
// ===== library: MasterCopy "GB2312_TO_UTF8" =====

// folder: FB/GB2312_UTF8

FUNCTION_BLOCK "GB2312_TO_UTF8"   // FB8, SCL
{ S7_Optimized_Access := 'TRUE' }
VERSION : 0.1
   VAR_INPUT
      GB2312 : String[254];
   END_VAR
   VAR_OUTPUT
      UTF8 : String[254];
   END_VAR
   VAR
      g_u : "GB2_TO_UNI";
      u_u8 : "UNI_TO_UTF8";
   END_VAR
   VAR_TEMP
      i : UDInt;
      j : UDInt;
      lenGB2 : Int;
      tempword : Word;
      tempstr : String[4];
   END_VAR
BEGIN
   #UTF8 := '';
   #lenGB2 := LEN(#GB2312);
   IF #lenGB2 > 0 THEN
       #j := 1;
       FOR #i := 1 TO INT_TO_UDINT(#lenGB2) DO
           IF #i = #j THEN
               IF BYTE_TO_WORD(#GB2312[#i]) < 16#0080 THEN
                   #tempword := BYTE_TO_WORD(#GB2312[#i]);
                   #j := #j + 1;
               ELSE
                   #tempword := BYTE_TO_WORD(#GB2312[#i]);
                   #tempword := SHL(IN := #tempword, N := 8);
                   #tempword := #tempword OR BYTE_TO_WORD(#GB2312[#i + 1]);
                   #j := #j + 2;
               END_IF;
               #g_u(GB2312 := #tempword,
                    UNICODE => #tempword);
               #u_u8(UNICODE := #tempword,
                     UTF8 => #tempstr);
               #UTF8 := CONCAT(IN1 := #UTF8, IN2 := #tempstr);
           END_IF;
       END_FOR;
   END_IF;
END_FUNCTION_BLOCK

// ===== library: MasterCopy "UTF8_TO_GB2312" =====

// folder: FB/GB2312_UTF8

FUNCTION_BLOCK "UTF8_TO_GB2312"   // FB10, SCL
{ S7_Optimized_Access := 'TRUE' }
VERSION : 0.1
   VAR_INPUT
      UTF8 : String[254];
   END_VAR
   VAR_OUTPUT
      GB2312 : String[254];
   END_VAR
   VAR
      u8_u : "UTF8_TO_UNI";
      u_g : "UNI_TO_GB2";
   END_VAR
   VAR_TEMP
      i : Int;
      j : Int;
      lenUTF8 : Int;
      tempword : Word;
      tempstr : String[5];
   END_VAR
BEGIN
   #GB2312 := '';
   #tempstr := '0000';
   #lenUTF8 := LEN(#UTF8);
   IF #lenUTF8 > 0 THEN
       #j := 1;
       FOR #i := 1 TO #lenUTF8 DO
           IF #i = #j THEN
               IF BYTE_TO_WORD(#UTF8[#i]) < 16#0080 THEN
                   #tempstr := MID(IN := #UTF8, L := 1, P := #i);
                   #j := #j + 1;
               ELSIF BYTE_TO_WORD(#UTF8[#i]) >= 16#C0 AND BYTE_TO_WORD(#UTF8[#i]) < 16#E0 THEN
                   #tempstr := MID(IN := #UTF8, L := 2, P := #i);
                   #j := #j + 2;
               ELSIF BYTE_TO_WORD(#UTF8[#i]) >= 16#E0 AND BYTE_TO_WORD(#UTF8[#i]) < 16#F0 THEN
                   #tempstr := MID(IN := #UTF8, L := 3, P := #i);
                   #j := #j + 3;
               ELSIF BYTE_TO_WORD(#UTF8[#i]) >= 16#F0 AND BYTE_TO_WORD(#UTF8[#i]) < 16#F8 THEN
                   #tempstr := MID(IN := #UTF8, L := 4, P := #i);
                   #j := #j + 4;
               END_IF;
               IF BYTE_TO_WORD(#UTF8[#i]) >= 16#0080 THEN
                   #u8_u(UTF8 := #tempstr,
                         UNICODE => #tempword);
                   #u_g(UNICODE := #tempword,
                        GB2312 => #tempword);
                   #tempstr[2] := WORD_TO_BYTE(#tempword AND 16#FF);
                   #tempstr[1] := WORD_TO_BYTE(SHR(IN := #tempword, N := 8) AND 16#FF);
                   #tempstr := LEFT(IN := #tempstr, L := 2);
               END_IF;
               #GB2312 := CONCAT(IN1 := #GB2312, IN2 := #tempstr);
           END_IF;
       END_FOR;
   END_IF;
END_FUNCTION_BLOCK

// ===== library: MasterCopy "GB2312_TO_UTF16" =====

// folder: FB/GB2312_UTF16

FUNCTION_BLOCK "GB2312_TO_UTF16"   // FB13, SCL
{ S7_Optimized_Access := 'TRUE' }
VERSION : 0.1
   VAR_INPUT
      GB2312 : String[254];
   END_VAR
   VAR_OUTPUT
      UTF16 : WString;
   END_VAR
   VAR
      g_u : "GB2_TO_UNI";
   END_VAR
   VAR_TEMP
      i : UDInt;
      j : UDInt;
      lenGB2 : Int;
      tempword : Word;
      tempWstr : WString[4];
   END_VAR
BEGIN
   #UTF16 := WSTRING#'';
   #tempWstr := WSTRING#'0000';
   #lenGB2 := LEN(#GB2312);
   IF #lenGB2 > 0 THEN
       #j := 1;
       FOR #i := 1 TO INT_TO_UDINT(#lenGB2) DO
           IF #i = #j THEN
               IF BYTE_TO_WORD(#GB2312[#i]) < 16#0080 THEN
                   #tempword := BYTE_TO_WORD(#GB2312[#i]);
                   #j := #j + 1;
               ELSE
                   #tempword := BYTE_TO_WORD(#GB2312[#i]);
                   #tempword := SHL(IN := #tempword, N := 8);
                   #tempword := #tempword OR BYTE_TO_WORD(#GB2312[#i + 1]);
                   #j := #j + 2;
               END_IF;
               #g_u(GB2312 := #tempword,
                    UNICODE => #tempword);
               #tempWstr[1] := #tempword;
               #tempWstr := LEFT(IN := #tempWstr, L := 1);
               #UTF16 := CONCAT(IN1 := #UTF16, IN2 := #tempWstr);
           END_IF;
       END_FOR;
   END_IF;
END_FUNCTION_BLOCK

// ===== library: MasterCopy "UTF16_TO_GB2312" =====

// folder: FB/GB2312_UTF16

FUNCTION_BLOCK "UTF16_TO_GB2312"   // FB11, SCL
{ S7_Optimized_Access := 'TRUE' }
VERSION : 0.1
   VAR_INPUT
      UTF16 : WString;
   END_VAR
   VAR_OUTPUT
      GB2312 : String[254];
   END_VAR
   VAR
      u_g : "UNI_TO_GB2";
   END_VAR
   VAR_TEMP
      i : Int;
      j : Int;
      lenUTF16 : Int;
      tempword : Word;
      tempstr : String[5];
   END_VAR
BEGIN
   #GB2312 := '';
   #tempstr := '0000';
   #lenUTF16 := LEN(#UTF16);
   IF #lenUTF16 > 0 THEN
       #j := 1;
       FOR #i := 1 TO #lenUTF16 DO
           #tempword := WCHAR_TO_WORD(#UTF16[#i]);
           IF #tempword < 16#0080 THEN
               #tempstr[1] := WORD_TO_BYTE(#tempword);
               #tempstr := LEFT(IN := #tempstr, L := 1);
           END_IF;
           IF #tempword >= 16#0080 THEN
               #u_g(UNICODE := #tempword,
                    GB2312 => #tempword);
               #tempstr[2] := WORD_TO_BYTE(#tempword AND 16#FF);
               #tempstr[1] := WORD_TO_BYTE(SHR(IN := #tempword, N := 8) AND 16#FF);
               #tempstr := LEFT(IN := #tempstr, L := 2);
           END_IF;
           #GB2312 := CONCAT(IN1 := #GB2312, IN2 := #tempstr);
       END_FOR;
   END_IF;
END_FUNCTION_BLOCK

// ===== library: MasterCopy "WStr_TO_Str_x4" =====

// folder: FB/GB2312_UTF16

FUNCTION_BLOCK "WStr_TO_Str_x4"   // FB12, SCL
{ S7_Optimized_Access := 'TRUE' }
VERSION : 0.1
   VAR_INPUT
      X0_Wstr : WString;
      X1_Wstr : WString;
      X2_Wstr : WString;
      X3_Wstr : WString;
   END_VAR
   VAR_OUTPUT
      X0_Str : String;
      X1_Str : String;
      X2_Str : String;
      X3_Str : String;
   END_VAR
   VAR
      U16_gb2 : "UTF16_TO_GB2312";
   END_VAR
   VAR_TEMP
      i : Int;
      j : Int;
      lenUTF16 : Int;
      tempword : Word;
      tempstr : String[5];
   END_VAR
BEGIN
   #U16_gb2(UTF16 := #X0_Wstr,
            GB2312 => #X0_Str);
   #U16_gb2(UTF16 := #X1_Wstr,
            GB2312 => #X1_Str);
   #U16_gb2(UTF16 := #X2_Wstr,
            GB2312 => #X2_Str);
   #U16_gb2(UTF16 := #X3_Wstr,
            GB2312 => #X3_Str);
END_FUNCTION_BLOCK

// ===== library: MasterCopy "UTF8_TO_GBK" =====

// folder: FB/GBK_UTF8

FUNCTION_BLOCK "UTF8_TO_GBK"   // FB6, SCL
{ S7_Optimized_Access := 'TRUE' }
VERSION : 0.1
   VAR_INPUT
      UTF8 : String[254];
   END_VAR
   VAR_OUTPUT
      GBK : String[254];
   END_VAR
   VAR
      u8_u : "UTF8_TO_UNI";
      u_g : "UNI_TO_GBK";
   END_VAR
   VAR_TEMP
      i : Int;
      j : Int;
      lenUTF8 : Int;
      tempword : Word;
      tempstr : String[5];
   END_VAR
BEGIN
   #GBK := '';
   #tempstr := '0000';
   #lenUTF8 := LEN(#UTF8);
   IF #lenUTF8 > 0 THEN
       #j := 1;
       FOR #i := 1 TO #lenUTF8 DO
           IF #i = #j THEN
               IF BYTE_TO_WORD(#UTF8[#i]) < 16#0080 THEN
                   #tempstr := MID(IN := #UTF8, L := 1, P := #i);
                   #j := #j + 1;
               ELSIF BYTE_TO_WORD(#UTF8[#i]) >= 16#C0 AND BYTE_TO_WORD(#UTF8[#i]) < 16#E0 THEN
                   #tempstr := MID(IN := #UTF8, L := 2, P := #i);
                   #j := #j + 2;
               ELSIF BYTE_TO_WORD(#UTF8[#i]) >= 16#E0 AND BYTE_TO_WORD(#UTF8[#i]) < 16#F0 THEN
                   #tempstr := MID(IN := #UTF8, L := 3, P := #i);
                   #j := #j + 3;
               ELSIF BYTE_TO_WORD(#UTF8[#i]) >= 16#F0 AND BYTE_TO_WORD(#UTF8[#i]) < 16#F8 THEN
                   #tempstr := MID(IN := #UTF8, L := 4, P := #i);
                   #j := #j + 4;
               END_IF;
               IF BYTE_TO_WORD(#UTF8[#i]) >= 16#0080 THEN
                   #u8_u(UTF8 := #tempstr,
                         UNICODE => #tempword);
                   #u_g(UNICODE := #tempword,
                        GBK => #tempword);
                   #tempstr[2] := WORD_TO_BYTE(#tempword AND 16#FF);
                   #tempstr[1] := WORD_TO_BYTE(SHR(IN := #tempword, N := 8) AND 16#FF);
                   #tempstr := LEFT(IN := #tempstr, L := 2);
               END_IF;
               #GBK := CONCAT(IN1 := #GBK, IN2 := #tempstr);
           END_IF;
       END_FOR;
   END_IF;
END_FUNCTION_BLOCK

// ===== library: MasterCopy "GBK_TO_UTF8" =====

// folder: FB/GBK_UTF8

FUNCTION_BLOCK "GBK_TO_UTF8"   // FB5, SCL
{ S7_Optimized_Access := 'TRUE' }
VERSION : 0.1
   VAR_INPUT
      GBK : String[254];
   END_VAR
   VAR_OUTPUT
      UTF8 : String[254];
   END_VAR
   VAR
      g_u : "GBK_TO_UNI";
      u_u8 : "UNI_TO_UTF8";
   END_VAR
   VAR_TEMP
      i : UDInt;
      j : UDInt;
      lenGBK : Int;
      tempword : Word;
      tempstr : String[4];
   END_VAR
BEGIN
   #UTF8 := '';
   #lenGBK := LEN(#GBK);
   IF #lenGBK > 0 THEN
       #j := 1;
       FOR #i := 1 TO INT_TO_UDINT(#lenGBK) DO
           IF #i = #j THEN
               IF BYTE_TO_WORD(#GBK[#i]) < 16#0080 THEN
                   #tempword := BYTE_TO_WORD(#GBK[#i]);
                   #j := #j + 1;
               ELSE
                   #tempword := BYTE_TO_WORD(#GBK[#i]);
                   #tempword := SHL(IN := #tempword, N:=8);
                   #tempword := #tempword OR BYTE_TO_WORD(#GBK[#i + 1]);
                   #j := #j + 2;
               END_IF;
               #g_u(GBK := #tempword,
                    UNICODE => #tempword);
               #u_u8(UNICODE := #tempword,
                     UTF8 => #tempstr);
               #UTF8 := CONCAT(IN1 := #UTF8, IN2 := #tempstr);
           END_IF;
       END_FOR;
   END_IF;
END_FUNCTION_BLOCK

// ===== library: MasterCopy "GB2_TO_UNI" =====

// folder: FB/UNICODE_FB

FUNCTION_BLOCK "GB2_TO_UNI"   // FB7, SCL
{ S7_Optimized_Access := 'TRUE' }
VERSION : 0.1
   VAR_INPUT
      GB2312 : Word;
   END_VAR
   VAR_OUTPUT
      UNICODE : Word;
   END_VAR
   VAR
      GB2 : Array[0..7480] of Word;
      UNI : Array[0..7480] of Word;
   END_VAR
   VAR_TEMP
      i : UDInt;
      j : UDInt;
      li : UDInt;
      hi : UDInt;
   END_VAR
   // GB2[0] := 16#A1A1;
   // GB2[1] := 16#A1A2;
   // GB2[2] := 16#A1A3;
   // GB2[3] := 16#A1A4;
   // GB2[4] := 16#A1A5;
   // GB2[5] := 16#A1A6;
   // GB2[6] := 16#A1A7;
   // GB2[7] := 16#A1A8;
   // GB2[8] := 16#A1A9;
   // GB2[9] := 16#A1AA;
   // GB2[10] := 16#A1AB;
   // GB2[11] := 16#A1AC;
   // GB2[12] := 16#A1AD;
   // GB2[13] := 16#A1AE;
   // GB2[14] := 16#A1AF;
   // GB2[15] := 16#A1B0;
   // GB2[16] := 16#A1B1;
   // GB2[17] := 16#A1B2;
   // GB2[18] := 16#A1B3;
   // GB2[19] := 16#A1B4;
   // GB2[20] := 16#A1B5;
   // GB2[21] := 16#A1B6;
   // GB2[22] := 16#A1B7;
   // GB2[23] := 16#A1B8;
   // GB2[24] := 16#A1B9;
   // GB2[25] := 16#A1BA;
   // GB2[26] := 16#A1BB;
   // GB2[27] := 16#A1BC;
   // GB2[28] := 16#A1BD;
   // GB2[29] := 16#A1BE;
   // GB2[30] := 16#A1BF;
   // GB2[31] := 16#A1C0;
   // GB2[32] := 16#A1C1;
   // GB2[33] := 16#A1C2;
   // GB2[34] := 16#A1C3;
   // GB2[35] := 16#A1C4;
   // GB2[36] := 16#A1C5;
   // GB2[37] := 16#A1C6;
   // GB2[38] := 16#A1C7;
   // GB2[39] := 16#A1C8;
   // GB2[40] := 16#A1C9;
   // GB2[41] := 16#A1CA;
   // GB2[42] := 16#A1CB;
   // GB2[43] := 16#A1CC;
   // GB2[44] := 16#A1CD;
   // GB2[45] := 16#A1CE;
   // GB2[46] := 16#A1CF;
   // GB2[47] := 16#A1D0;
   // GB2[48] := 16#A1D1;
   // GB2[49] := 16#A1D2;
   // GB2[50] := 16#A1D3;
   // GB2[51] := 16#A1D4;
   // GB2[52] := 16#A1D5;
   // GB2[53] := 16#A1D6;
   // GB2[54] := 16#A1D7;
   // GB2[55] := 16#A1D8;
   // GB2[56] := 16#A1D9;
   // GB2[57] := 16#A1DA;
   // GB2[58] := 16#A1DB;
   // GB2[59] := 16#A1DC;
   // GB2[60] := 16#A1DD;
   // GB2[61] := 16#A1DE;
   // GB2[62] := 16#A1DF;
   // GB2[63] := 16#A1E0;
   // GB2[64] := 16#A1E1;
   // GB2[65] := 16#A1E2;
   // GB2[66] := 16#A1E3;
   // GB2[67] := 16#A1E4;
   // GB2[68] := 16#A1E5;
   // GB2[69] := 16#A1E6;
   // GB2[70] := 16#A1E7;
   // GB2[71] := 16#A1E8;
   // GB2[72] := 16#A1E9;
   // GB2[73] := 16#A1EA;
   // GB2[74] := 16#A1EB;
   // GB2[75] := 16#A1EC;
   // GB2[76] := 16#A1ED;
   // GB2[77] := 16#A1EE;
   // GB2[78] := 16#A1EF;
   // GB2[79] := 16#A1F0;
   // GB2[80] := 16#A1F1;
   // GB2[81] := 16#A1F2;
   // GB2[82] := 16#A1F3;
   // GB2[83] := 16#A1F4;
   // GB2[84] := 16#A1F5;
   // GB2[85] := 16#A1F6;
   // GB2[86] := 16#A1F7;
   // GB2[87] := 16#A1F8;
   // GB2[88] := 16#A1F9;
   // GB2[89] := 16#A1FA;
   // GB2[90] := 16#A1FB;
   // GB2[91] := 16#A1FC;
   // GB2[92] := 16#A1FD;
   // GB2[93] := 16#A1FE;
   // GB2[94] := 16#A2A1;
   // GB2[95] := 16#A2A2;
   // GB2[96] := 16#A2A3;
   // GB2[97] := 16#A2A4;
   // GB2[98] := 16#A2A5;
   // GB2[99] := 16#A2A6;
   // GB2[100] := 16#A2A7;
   // GB2[101] := 16#A2A8;
   // GB2[102] := 16#A2A9;
   // GB2[103] := 16#A2AA;
   // GB2[104] := 16#A2B1;
   // GB2[105] := 16#A2B2;
   // GB2[106] := 16#A2B3;
   // GB2[107] := 16#A2B4;
   // GB2[108] := 16#A2B5;
   // GB2[109] := 16#A2B6;
   // GB2[110] := 16#A2B7;
   // GB2[111] := 16#A2B8;
   // GB2[112] := 16#A2B9;
   // GB2[113] := 16#A2BA;
   // GB2[114] := 16#A2BB;
   // GB2[115] := 16#A2BC;
   // GB2[116] := 16#A2BD;
   // GB2[117] := 16#A2BE;
   // GB2[118] := 16#A2BF;
   // GB2[119] := 16#A2C0;
   // GB2[120] := 16#A2C1;
   // GB2[121] := 16#A2C2;
   // GB2[122] := 16#A2C3;
   // GB2[123] := 16#A2C4;
   // GB2[124] := 16#A2C5;
   // GB2[125] := 16#A2C6;
   // GB2[126] := 16#A2C7;
   // GB2[127] := 16#A2C8;
   // GB2[128] := 16#A2C9;
   // GB2[129] := 16#A2CA;
   // GB2[130] := 16#A2CB;
   // GB2[131] := 16#A2CC;
   // GB2[132] := 16#A2CD;
   // GB2[133] := 16#A2CE;
   // GB2[134] := 16#A2CF;
   // GB2[135] := 16#A2D0;
   // GB2[136] := 16#A2D1;
   // GB2[137] := 16#A2D2;
   // GB2[138] := 16#A2D3;
   // GB2[139] := 16#A2D4;
   // GB2[140] := 16#A2D5;
   // GB2[141] := 16#A2D6;
   // GB2[142] := 16#A2D7;
   // GB2[143] := 16#A2D8;
   // GB2[144] := 16#A2D9;
   // GB2[145] := 16#A2DA;
   // GB2[146] := 16#A2DB;
   // GB2[147] := 16#A2DC;
   // GB2[148] := 16#A2DD;
   // GB2[149] := 16#A2DE;
   // GB2[150] := 16#A2DF;
   // GB2[151] := 16#A2E0;
   // GB2[152] := 16#A2E1;
   // GB2[153] := 16#A2E2;
   // GB2[154] := 16#A2E5;
   // GB2[155] := 16#A2E6;
   // GB2[156] := 16#A2E7;
   // GB2[157] := 16#A2E8;
   // GB2[158] := 16#A2E9;
   // GB2[159] := 16#A2EA;
   // GB2[160] := 16#A2EB;
   // GB2[161] := 16#A2EC;
   // GB2[162] := 16#A2ED;
   // GB2[163] := 16#A2EE;
   // GB2[164] := 16#A2F1;
   // GB2[165] := 16#A2F2;
   // GB2[166] := 16#A2F3;
   // GB2[167] := 16#A2F4;
   // GB2[168] := 16#A2F5;
   // GB2[169] := 16#A2F6;
   // GB2[170] := 16#A2F7;
   // GB2[171] := 16#A2F8;
   // GB2[172] := 16#A2F9;
   // GB2[173] := 16#A2FA;
   // GB2[174] := 16#A2FB;
   // GB2[175] := 16#A2FC;
   // GB2[176] := 16#A3A1;
   // GB2[177] := 16#A3A2;
   // GB2[178] := 16#A3A3;
   // GB2[179] := 16#A3A4;
   // GB2[180] := 16#A3A5;
   // GB2[181] := 16#A3A6;
   // GB2[182] := 16#A3A7;
   // GB2[183] := 16#A3A8;
   // GB2[184] := 16#A3A9;
   // GB2[185] := 16#A3AA;
   // GB2[186] := 16#A3AB;
   // GB2[187] := 16#A3AC;
   // GB2[188] := 16#A3AD;
   // GB2[189] := 16#A3AE;
   // GB2[190] := 16#A3AF;
   // GB2[191] := 16#A3B0;
   // GB2[192] := 16#A3B1;
   // GB2[193] := 16#A3B2;
   // GB2[194] := 16#A3B3;
   // GB2[195] := 16#A3B4;
   // GB2[196] := 16#A3B5;
   // GB2[197] := 16#A3B6;
   // GB2[198] := 16#A3B7;
   // GB2[199] := 16#A3B8;
   // GB2[200] := 16#A3B9;
   // GB2[201] := 16#A3BA;
   // GB2[202] := 16#A3BB;
   // GB2[203] := 16#A3BC;
   // GB2[204] := 16#A3BD;
   // GB2[205] := 16#A3BE;
   // GB2[206] := 16#A3BF;
   // GB2[207] := 16#A3C0;
   // GB2[208] := 16#A3C1;
   // GB2[209] := 16#A3C2;
   // GB2[210] := 16#A3C3;
   // GB2[211] := 16#A3C4;
   // GB2[212] := 16#A3C5;
   // GB2[213] := 16#A3C6;
   // GB2[214] := 16#A3C7;
   // GB2[215] := 16#A3C8;
   // GB2[216] := 16#A3C9;
   // GB2[217] := 16#A3CA;
   // GB2[218] := 16#A3CB;
   // GB2[219] := 16#A3CC;
   // GB2[220] := 16#A3CD;
   // GB2[221] := 16#A3CE;
   // GB2[222] := 16#A3CF;
   // GB2[223] := 16#A3D0;
   // GB2[224] := 16#A3D1;
   // GB2[225] := 16#A3D2;
   // GB2[226] := 16#A3D3;
   // GB2[227] := 16#A3D4;
   // GB2[228] := 16#A3D5;
   // GB2[229] := 16#A3D6;
   // GB2[230] := 16#A3D7;
   // GB2[231] := 16#A3D8;
   // GB2[232] := 16#A3D9;
   // GB2[233] := 16#A3DA;
   // GB2[234] := 16#A3DB;
   // GB2[235] := 16#A3DC;
   // GB2[236] := 16#A3DD;
   // GB2[237] := 16#A3DE;
   // GB2[238] := 16#A3DF;
   // GB2[239] := 16#A3E0;
   // GB2[240] := 16#A3E1;
   // GB2[241] := 16#A3E2;
   // GB2[242] := 16#A3E3;
   // GB2[243] := 16#A3E4;
   // GB2[244] := 16#A3E5;
   // GB2[245] := 16#A3E6;
   // GB2[246] := 16#A3E7;
   // GB2[247] := 16#A3E8;
   // GB2[248] := 16#A3E9;
   // GB2[249] := 16#A3EA;
   // GB2[250] := 16#A3EB;
   // GB2[251] := 16#A3EC;
   // GB2[252] := 16#A3ED;
   // GB2[253] := 16#A3EE;
   // GB2[254] := 16#A3EF;
   // GB2[255] := 16#A3F0;
   // GB2[256] := 16#A3F1;
   // GB2[257] := 16#A3F2;
   // GB2[258] := 16#A3F3;
   // GB2[259] := 16#A3F4;
   // GB2[260] := 16#A3F5;
   // GB2[261] := 16#A3F6;
   // GB2[262] := 16#A3F7;
   // GB2[263] := 16#A3F8;
   // GB2[264] := 16#A3F9;
   // GB2[265] := 16#A3FA;
   // GB2[266] := 16#A3FB;
   // GB2[267] := 16#A3FC;
   // GB2[268] := 16#A3FD;
   // GB2[269] := 16#A3FE;
   // GB2[270] := 16#A4A1;
   // GB2[271] := 16#A4A2;
   // GB2[272] := 16#A4A3;
   // GB2[273] := 16#A4A4;
   // GB2[274] := 16#A4A5;
   // GB2[275] := 16#A4A6;
   // GB2[276] := 16#A4A7;
   // GB2[277] := 16#A4A8;
   // GB2[278] := 16#A4A9;
   // GB2[279] := 16#A4AA;
   // GB2[280] := 16#A4AB;
   // GB2[281] := 16#A4AC;
   // GB2[282] := 16#A4AD;
   // GB2[283] := 16#A4AE;
   // GB2[284] := 16#A4AF;
   // GB2[285] := 16#A4B0;
   // GB2[286] := 16#A4B1;
   // GB2[287] := 16#A4B2;
   // GB2[288] := 16#A4B3;
   // GB2[289] := 16#A4B4;
   // GB2[290] := 16#A4B5;
   // GB2[291] := 16#A4B6;
   // GB2[292] := 16#A4B7;
   // GB2[293] := 16#A4B8;
   // GB2[294] := 16#A4B9;
   // GB2[295] := 16#A4BA;
   // GB2[296] := 16#A4BB;
   // GB2[297] := 16#A4BC;
   // GB2[298] := 16#A4BD;
   // GB2[299] := 16#A4BE;
   // GB2[300] := 16#A4BF;
   // GB2[301] := 16#A4C0;
   // GB2[302] := 16#A4C1;
   // GB2[303] := 16#A4C2;
   // GB2[304] := 16#A4C3;
   // GB2[305] := 16#A4C4;
   // GB2[306] := 16#A4C5;
   // GB2[307] := 16#A4C6;
   // GB2[308] := 16#A4C7;
   // GB2[309] := 16#A4C8;
   // GB2[310] := 16#A4C9;
   // GB2[311] := 16#A4CA;
   // GB2[312] := 16#A4CB;
   // GB2[313] := 16#A4CC;
   // GB2[314] := 16#A4CD;
   // GB2[315] := 16#A4CE;
   // GB2[316] := 16#A4CF;
   // GB2[317] := 16#A4D0;
   // GB2[318] := 16#A4D1;
   // GB2[319] := 16#A4D2;
   // GB2[320] := 16#A4D3;
   // GB2[321] := 16#A4D4;
   // GB2[322] := 16#A4D5;
   // GB2[323] := 16#A4D6;
   // GB2[324] := 16#A4D7;
   // GB2[325] := 16#A4D8;
   // GB2[326] := 16#A4D9;
   // GB2[327] := 16#A4DA;
   // GB2[328] := 16#A4DB;
   // GB2[329] := 16#A4DC;
   // GB2[330] := 16#A4DD;
   // GB2[331] := 16#A4DE;
   // GB2[332] := 16#A4DF;
   // GB2[333] := 16#A4E0;
   // GB2[334] := 16#A4E1;
   // GB2[335] := 16#A4E2;
   // GB2[336] := 16#A4E3;
   // GB2[337] := 16#A4E4;
   // GB2[338] := 16#A4E5;
   // GB2[339] := 16#A4E6;
   // GB2[340] := 16#A4E7;
   // GB2[341] := 16#A4E8;
   // GB2[342] := 16#A4E9;
   // GB2[343] := 16#A4EA;
   // GB2[344] := 16#A4EB;
   // GB2[345] := 16#A4EC;
   // GB2[346] := 16#A4ED;
   // GB2[347] := 16#A4EE;
   // GB2[348] := 16#A4EF;
   // GB2[349] := 16#A4F0;
   // GB2[350] := 16#A4F1;
   // GB2[351] := 16#A4F2;
   // GB2[352] := 16#A4F3;
   // GB2[353] := 16#A5A1;
   // GB2[354] := 16#A5A2;
   // GB2[355] := 16#A5A3;
   // GB2[356] := 16#A5A4;
   // GB2[357] := 16#A5A5;
   // GB2[358] := 16#A5A6;
   // GB2[359] := 16#A5A7;
   // GB2[360] := 16#A5A8;
   // GB2[361] := 16#A5A9;
   // GB2[362] := 16#A5AA;
   // GB2[363] := 16#A5AB;
   // GB2[364] := 16#A5AC;
   // GB2[365] := 16#A5AD;
   // GB2[366] := 16#A5AE;
   // GB2[367] := 16#A5AF;
   // GB2[368] := 16#A5B0;
   // GB2[369] := 16#A5B1;
   // GB2[370] := 16#A5B2;
   // GB2[371] := 16#A5B3;
   // GB2[372] := 16#A5B4;
   // GB2[373] := 16#A5B5;
   // GB2[374] := 16#A5B6;
   // GB2[375] := 16#A5B7;
   // GB2[376] := 16#A5B8;
   // GB2[377] := 16#A5B9;
   // GB2[378] := 16#A5BA;
   // GB2[379] := 16#A5BB;
   // GB2[380] := 16#A5BC;
   // GB2[381] := 16#A5BD;
   // GB2[382] := 16#A5BE;
   // GB2[383] := 16#A5BF;
   // GB2[384] := 16#A5C0;
   // GB2[385] := 16#A5C1;
   // GB2[386] := 16#A5C2;
   // GB2[387] := 16#A5C3;
   // GB2[388] := 16#A5C4;
   // GB2[389] := 16#A5C5;
   // GB2[390] := 16#A5C6;
   // GB2[391] := 16#A5C7;
   // GB2[392] := 16#A5C8;
   // GB2[393] := 16#A5C9;
   // GB2[394] := 16#A5CA;
   // GB2[395] := 16#A5CB;
   // GB2[396] := 16#A5CC;
   // GB2[397] := 16#A5CD;
   // GB2[398] := 16#A5CE;
   // GB2[399] := 16#A5CF;
   // GB2[400] := 16#A5D0;
   // GB2[401] := 16#A5D1;
   // GB2[402] := 16#A5D2;
   // GB2[403] := 16#A5D3;
   // GB2[404] := 16#A5D4;
   // GB2[405] := 16#A5D5;
   // GB2[406] := 16#A5D6;
   // GB2[407] := 16#A5D7;
   // GB2[408] := 16#A5D8;
   // GB2[409] := 16#A5D9;
   // GB2[410] := 16#A5DA;
   // GB2[411] := 16#A5DB;
   // GB2[412] := 16#A5DC;
   // GB2[413] := 16#A5DD;
   // GB2[414] := 16#A5DE;
   // GB2[415] := 16#A5DF;
   // GB2[416] := 16#A5E0;
   // GB2[417] := 16#A5E1;
   // GB2[418] := 16#A5E2;
   // GB2[419] := 16#A5E3;
   // GB2[420] := 16#A5E4;
   // GB2[421] := 16#A5E5;
   // GB2[422] := 16#A5E6;
   // GB2[423] := 16#A5E7;
   // GB2[424] := 16#A5E8;
   // GB2[425] := 16#A5E9;
   // GB2[426] := 16#A5EA;
   // GB2[427] := 16#A5EB;
   // GB2[428] := 16#A5EC;
   // GB2[429] := 16#A5ED;
   // GB2[430] := 16#A5EE;
   // GB2[431] := 16#A5EF;
   // GB2[432] := 16#A5F0;
   // GB2[433] := 16#A5F1;
   // GB2[434] := 16#A5F2;
   // GB2[435] := 16#A5F3;
   // GB2[436] := 16#A5F4;
   // GB2[437] := 16#A5F5;
   // GB2[438] := 16#A5F6;
   // GB2[439] := 16#A6A1;
   // GB2[440] := 16#A6A2;
   // GB2[441] := 16#A6A3;
   // GB2[442] := 16#A6A4;
   // GB2[443] := 16#A6A5;
   // GB2[444] := 16#A6A6;
   // GB2[445] := 16#A6A7;
   // GB2[446] := 16#A6A8;
   // GB2[447] := 16#A6A9;
   // GB2[448] := 16#A6AA;
   // GB2[449] := 16#A6AB;
   // GB2[450] := 16#A6AC;
   // GB2[451] := 16#A6AD;
   // GB2[452] := 16#A6AE;
   // GB2[453] := 16#A6AF;
   // GB2[454] := 16#A6B0;
   // GB2[455] := 16#A6B1;
   // GB2[456] := 16#A6B2;
   // GB2[457] := 16#A6B3;
   // GB2[458] := 16#A6B4;
   // GB2[459] := 16#A6B5;
   // GB2[460] := 16#A6B6;
   // GB2[461] := 16#A6B7;
   // GB2[462] := 16#A6B8;
   // GB2[463] := 16#A6C1;
   // GB2[464] := 16#A6C2;
   // GB2[465] := 16#A6C3;
   // GB2[466] := 16#A6C4;
   // GB2[467] := 16#A6C5;
   // GB2[468] := 16#A6C6;
   // GB2[469] := 16#A6C7;
   // GB2[470] := 16#A6C8;
   // GB2[471] := 16#A6C9;
   // GB2[472] := 16#A6CA;
   // GB2[473] := 16#A6CB;
   // GB2[474] := 16#A6CC;
   // GB2[475] := 16#A6CD;
   // GB2[476] := 16#A6CE;
   // GB2[477] := 16#A6CF;
   // GB2[478] := 16#A6D0;
   // GB2[479] := 16#A6D1;
   // GB2[480] := 16#A6D2;
   // GB2[481] := 16#A6D3;
   // GB2[482] := 16#A6D4;
   // GB2[483] := 16#A6D5;
   // GB2[484] := 16#A6D6;
   // GB2[485] := 16#A6D7;
   // GB2[486] := 16#A6D8;
   // GB2[487] := 16#A6E0;
   // GB2[488] := 16#A6E1;
   // GB2[489] := 16#A6E2;
   // GB2[490] := 16#A6E3;
   // GB2[491] := 16#A6E4;
   // GB2[492] := 16#A6E5;
   // GB2[493] := 16#A6E6;
   // GB2[494] := 16#A6E7;
   // GB2[495] := 16#A6E8;
   // GB2[496] := 16#A6E9;
   // GB2[497] := 16#A6EA;
   // GB2[498] := 16#A6EB;
   // GB2[499] := 16#A6EE;
   // GB2[500] := 16#A6EF;
   // GB2[501] := 16#A6F0;
   // GB2[502] := 16#A6F1;
   // GB2[503] := 16#A6F2;
   // GB2[504] := 16#A6F4;
   // GB2[505] := 16#A6F5;
   // GB2[506] := 16#A7A1;
   // GB2[507] := 16#A7A2;
   // GB2[508] := 16#A7A3;
   // GB2[509] := 16#A7A4;
   // GB2[510] := 16#A7A5;
   // GB2[511] := 16#A7A6;
   // GB2[512] := 16#A7A7;
   // GB2[513] := 16#A7A8;
   // GB2[514] := 16#A7A9;
   // GB2[515] := 16#A7AA;
   // GB2[516] := 16#A7AB;
   // GB2[517] := 16#A7AC;
   // GB2[518] := 16#A7AD;
   // GB2[519] := 16#A7AE;
   // GB2[520] := 16#A7AF;
   // GB2[521] := 16#A7B0;
   // GB2[522] := 16#A7B1;
   // GB2[523] := 16#A7B2;
   // GB2[524] := 16#A7B3;
   // GB2[525] := 16#A7B4;
   // GB2[526] := 16#A7B5;
   // GB2[527] := 16#A7B6;
   // GB2[528] := 16#A7B7;
   // GB2[529] := 16#A7B8;
   // GB2[530] := 16#A7B9;
   // GB2[531] := 16#A7BA;
   // GB2[532] := 16#A7BB;
   // GB2[533] := 16#A7BC;
   // GB2[534] := 16#A7BD;
   // GB2[535] := 16#A7BE;
   // GB2[536] := 16#A7BF;
   // GB2[537] := 16#A7C0;
   // GB2[538] := 16#A7C1;
   // GB2[539] := 16#A7D1;
   // GB2[540] := 16#A7D2;
   // GB2[541] := 16#A7D3;
   // GB2[542] := 16#A7D4;
   // GB2[543] := 16#A7D5;
   // GB2[544] := 16#A7D6;
   // GB2[545] := 16#A7D7;
   // GB2[546] := 16#A7D8;
   // GB2[547] := 16#A7D9;
   // GB2[548] := 16#A7DA;
   // GB2[549] := 16#A7DB;
   // GB2[550] := 16#A7DC;
   // GB2[551] := 16#A7DD;
   // GB2[552] := 16#A7DE;
   // GB2[553] := 16#A7DF;
   // GB2[554] := 16#A7E0;
   // GB2[555] := 16#A7E1;
   // GB2[556] := 16#A7E2;
   // GB2[557] := 16#A7E3;
   // GB2[558] := 16#A7E4;
   // GB2[559] := 16#A7E5;
   // GB2[560] := 16#A7E6;
   // GB2[561] := 16#A7E7;
   // GB2[562] := 16#A7E8;
   // GB2[563] := 16#A7E9;
   // GB2[564] := 16#A7EA;
   // GB2[565] := 16#A7EB;
   // GB2[566] := 16#A7EC;
   // GB2[567] := 16#A7ED;
   // GB2[568] := 16#A7EE;
   // GB2[569] := 16#A7EF;
   // GB2[570] := 16#A7F0;
   // GB2[571] := 16#A7F1;
   // GB2[572] := 16#A8A1;
   // GB2[573] := 16#A8A2;
   // GB2[574] := 16#A8A3;
   // GB2[575] := 16#A8A4;
   // GB2[576] := 16#A8A5;
   // GB2[577] := 16#A8A6;
   // GB2[578] := 16#A8A7;
   // GB2[579] := 16#A8A8;
   // GB2[580] := 16#A8A9;
   // GB2[581] := 16#A8AA;
   // GB2[582] := 16#A8AB;
   // GB2[583] := 16#A8AC;
   // GB2[584] := 16#A8AD;
   // GB2[585] := 16#A8AE;
   // GB2[586] := 16#A8AF;
   // GB2[587] := 16#A8B0;
   // GB2[588] := 16#A8B1;
   // GB2[589] := 16#A8B2;
   // GB2[590] := 16#A8B3;
   // GB2[591] := 16#A8B4;
   // GB2[592] := 16#A8B5;
   // GB2[593] := 16#A8B6;
   // GB2[594] := 16#A8B7;
   // GB2[595] := 16#A8B8;
   // GB2[596] := 16#A8B9;
   // GB2[597] := 16#A8BA;
   // GB2[598] := 16#A8BB;
   // GB2[599] := 16#A8BD;
   // GB2[600] := 16#A8BE;
   // GB2[601] := 16#A8C0;
   // GB2[602] := 16#A8C5;
   // GB2[603] := 16#A8C6;
   // GB2[604] := 16#A8C7;
   // GB2[605] := 16#A8C8;
   // GB2[606] := 16#A8C9;
   // GB2[607] := 16#A8CA;
   // GB2[608] := 16#A8CB;
   // GB2[609] := 16#A8CC;
   // GB2[610] := 16#A8CD;
   // GB2[611] := 16#A8CE;
   // GB2[612] := 16#A8CF;
   // GB2[613] := 16#A8D0;
   // GB2[614] := 16#A8D1;
   // GB2[615] := 16#A8D2;
   // GB2[616] := 16#A8D3;
   // GB2[617] := 16#A8D4;
   // GB2[618] := 16#A8D5;
   // GB2[619] := 16#A8D6;
   // GB2[620] := 16#A8D7;
   // GB2[621] := 16#A8D8;
   // GB2[622] := 16#A8D9;
   // GB2[623] := 16#A8DA;
   // GB2[624] := 16#A8DB;
   // GB2[625] := 16#A8DC;
   // GB2[626] := 16#A8DD;
   // GB2[627] := 16#A8DE;
   // GB2[628] := 16#A8DF;
   // GB2[629] := 16#A8E0;
   // GB2[630] := 16#A8E1;
   // GB2[631] := 16#A8E2;
   // GB2[632] := 16#A8E3;
   // GB2[633] := 16#A8E4;
   // GB2[634] := 16#A8E5;
   // GB2[635] := 16#A8E6;
   // GB2[636] := 16#A8E7;
   // GB2[637] := 16#A8E8;
   // GB2[638] := 16#A8E9;
   // GB2[639] := 16#A9A4;
   // GB2[640] := 16#A9A5;
   // GB2[641] := 16#A9A6;
   // GB2[642] := 16#A9A7;
   // GB2[643] := 16#A9A8;
   // GB2[644] := 16#A9A9;
   // GB2[645] := 16#A9AA;
   // GB2[646] := 16#A9AB;
   // GB2[647] := 16#A9AC;
   // GB2[648] := 16#A9AD;
   // GB2[649] := 16#A9AE;
   // GB2[650] := 16#A9AF;
   // GB2[651] := 16#A9B0;
   // GB2[652] := 16#A9B1;
   // GB2[653] := 16#A9B2;
   // GB2[654] := 16#A9B3;
   // GB2[655] := 16#A9B4;
   // GB2[656] := 16#A9B5;
   // GB2[657] := 16#A9B6;
   // GB2[658] := 16#A9B7;
   // GB2[659] := 16#A9B8;
   // GB2[660] := 16#A9B9;
   // GB2[661] := 16#A9BA;
   // GB2[662] := 16#A9BB;
   // GB2[663] := 16#A9BC;
   // GB2[664] := 16#A9BD;
   // GB2[665] := 16#A9BE;
   // GB2[666] := 16#A9BF;
   // GB2[667] := 16#A9C0;
   // GB2[668] := 16#A9C1;
   // GB2[669] := 16#A9C2;
   // GB2[670] := 16#A9C3;
   // GB2[671] := 16#A9C4;
   // GB2[672] := 16#A9C5;
   // GB2[673] := 16#A9C6;
   // GB2[674] := 16#A9C7;
   // GB2[675] := 16#A9C8;
   // GB2[676] := 16#A9C9;
   // GB2[677] := 16#A9CA;
   // GB2[678] := 16#A9CB;
   // GB2[679] := 16#A9CC;
   // GB2[680] := 16#A9CD;
   // GB2[681] := 16#A9CE;
   // GB2[682] := 16#A9CF;
   // GB2[683] := 16#A9D0;
   // GB2[684] := 16#A9D1;
   // GB2[685] := 16#A9D2;
   // GB2[686] := 16#A9D3;
   // GB2[687] := 16#A9D4;
   // GB2[688] := 16#A9D5;
   // GB2[689] := 16#A9D6;
   // GB2[690] := 16#A9D7;
   // GB2[691] := 16#A9D8;
   // GB2[692] := 16#A9D9;
   // GB2[693] := 16#A9DA;
   // GB2[694] := 16#A9DB;
   // GB2[695] := 16#A9DC;
   // GB2[696] := 16#A9DD;
   // GB2[697] := 16#A9DE;
   // GB2[698] := 16#A9DF;
   // GB2[699] := 16#A9E0;
   // GB2[700] := 16#A9E1;
   // GB2[701] := 16#A9E2;
   // GB2[702] := 16#A9E3;
   // GB2[703] := 16#A9E4;
   // GB2[704] := 16#A9E5;
   // GB2[705] := 16#A9E6;
   // GB2[706] := 16#A9E7;
   // GB2[707] := 16#A9E8;
   // GB2[708] := 16#A9E9;
   // GB2[709] := 16#A9EA;
   // GB2[710] := 16#A9EB;
   // GB2[711] := 16#A9EC;
   // GB2[712] := 16#A9ED;
   // GB2[713] := 16#A9EE;
   // GB2[714] := 16#A9EF;
   // GB2[715] := 16#B0A1;
   // GB2[716] := 16#B0A2;
   // GB2[717] := 16#B0A3;
   // GB2[718] := 16#B0A4;
   // GB2[719] := 16#B0A5;
   // GB2[720] := 16#B0A6;
   // GB2[721] := 16#B0A7;
   // GB2[722] := 16#B0A8;
   // GB2[723] := 16#B0A9;
   // GB2[724] := 16#B0AA;
   // GB2[725] := 16#B0AB;
   // GB2[726] := 16#B0AC;
   // GB2[727] := 16#B0AD;
   // GB2[728] := 16#B0AE;
   // GB2[729] := 16#B0AF;
   // GB2[730] := 16#B0B0;
   // GB2[731] := 16#B0B1;
   // GB2[732] := 16#B0B2;
   // GB2[733] := 16#B0B3;
   // GB2[734] := 16#B0B4;
   // GB2[735] := 16#B0B5;
   // GB2[736] := 16#B0B6;
   // GB2[737] := 16#B0B7;
   // GB2[738] := 16#B0B8;
   // GB2[739] := 16#B0B9;
   // GB2[740] := 16#B0BA;
   // GB2[741] := 16#B0BB;
   // GB2[742] := 16#B0BC;
   // GB2[743] := 16#B0BD;
   // GB2[744] := 16#B0BE;
   // GB2[745] := 16#B0BF;
   // GB2[746] := 16#B0C0;
   // GB2[747] := 16#B0C1;
   // GB2[748] := 16#B0C2;
   // GB2[749] := 16#B0C3;
   // GB2[750] := 16#B0C4;
   // GB2[751] := 16#B0C5;
   // GB2[752] := 16#B0C6;
   // GB2[753] := 16#B0C7;
   // GB2[754] := 16#B0C8;
   // GB2[755] := 16#B0C9;
   // GB2[756] := 16#B0CA;
   // GB2[757] := 16#B0CB;
   // GB2[758] := 16#B0CC;
   // GB2[759] := 16#B0CD;
   // GB2[760] := 16#B0CE;
   // GB2[761] := 16#B0CF;
   // GB2[762] := 16#B0D0;
   // GB2[763] := 16#B0D1;
   // GB2[764] := 16#B0D2;
   // GB2[765] := 16#B0D3;
   // GB2[766] := 16#B0D4;
   // GB2[767] := 16#B0D5;
   // GB2[768] := 16#B0D6;
   // GB2[769] := 16#B0D7;
   // GB2[770] := 16#B0D8;
   // GB2[771] := 16#B0D9;
   // GB2[772] := 16#B0DA;
   // GB2[773] := 16#B0DB;
   // GB2[774] := 16#B0DC;
   // GB2[775] := 16#B0DD;
   // GB2[776] := 16#B0DE;
   // GB2[777] := 16#B0DF;
   // GB2[778] := 16#B0E0;
   // GB2[779] := 16#B0E1;
   // GB2[780] := 16#B0E2;
   // GB2[781] := 16#B0E3;
   // GB2[782] := 16#B0E4;
   // GB2[783] := 16#B0E5;
   // GB2[784] := 16#B0E6;
   // GB2[785] := 16#B0E7;
   // GB2[786] := 16#B0E8;
   // GB2[787] := 16#B0E9;
   // GB2[788] := 16#B0EA;
   // GB2[789] := 16#B0EB;
   // GB2[790] := 16#B0EC;
   // GB2[791] := 16#B0ED;
   // GB2[792] := 16#B0EE;
   // GB2[793] := 16#B0EF;
   // GB2[794] := 16#B0F0;
   // GB2[795] := 16#B0F1;
   // GB2[796] := 16#B0F2;
   // GB2[797] := 16#B0F3;
   // GB2[798] := 16#B0F4;
   // GB2[799] := 16#B0F5;
   // GB2[800] := 16#B0F6;
   // GB2[801] := 16#B0F7;
   // GB2[802] := 16#B0F8;
   // GB2[803] := 16#B0F9;
   // GB2[804] := 16#B0FA;
   // GB2[805] := 16#B0FB;
   // GB2[806] := 16#B0FC;
   // GB2[807] := 16#B0FD;
   // GB2[808] := 16#B0FE;
   // GB2[809] := 16#B1A1;
   // GB2[810] := 16#B1A2;
   // GB2[811] := 16#B1A3;
   // GB2[812] := 16#B1A4;
   // GB2[813] := 16#B1A5;
   // GB2[814] := 16#B1A6;
   // GB2[815] := 16#B1A7;
   // GB2[816] := 16#B1A8;
   // GB2[817] := 16#B1A9;
   // GB2[818] := 16#B1AA;
   // GB2[819] := 16#B1AB;
   // GB2[820] := 16#B1AC;
   // GB2[821] := 16#B1AD;
   // GB2[822] := 16#B1AE;
   // GB2[823] := 16#B1AF;
   // GB2[824] := 16#B1B0;
   // GB2[825] := 16#B1B1;
   // GB2[826] := 16#B1B2;
   // GB2[827] := 16#B1B3;
   // GB2[828] := 16#B1B4;
   // GB2[829] := 16#B1B5;
   // GB2[830] := 16#B1B6;
   // GB2[831] := 16#B1B7;
   // GB2[832] := 16#B1B8;
   // GB2[833] := 16#B1B9;
   // GB2[834] := 16#B1BA;
   // GB2[835] := 16#B1BB;
   // GB2[836] := 16#B1BC;
   // GB2[837] := 16#B1BD;
   // GB2[838] := 16#B1BE;
   // GB2[839] := 16#B1BF;
   // GB2[840] := 16#B1C0;
   // GB2[841] := 16#B1C1;
   // GB2[842] := 16#B1C2;
   // GB2[843] := 16#B1C3;
   // GB2[844] := 16#B1C4;
   // GB2[845] := 16#B1C5;
   // GB2[846] := 16#B1C6;
   // GB2[847] := 16#B1C7;
   // GB2[848] := 16#B1C8;
   // GB2[849] := 16#B1C9;
   // GB2[850] := 16#B1CA;
   // GB2[851] := 16#B1CB;
   // GB2[852] := 16#B1CC;
   // GB2[853] := 16#B1CD;
   // GB2[854] := 16#B1CE;
   // GB2[855] := 16#B1CF;
   // GB2[856] := 16#B1D0;
   // GB2[857] := 16#B1D1;
   // GB2[858] := 16#B1D2;
   // GB2[859] := 16#B1D3;
   // GB2[860] := 16#B1D4;
   // GB2[861] := 16#B1D5;
   // GB2[862] := 16#B1D6;
   // GB2[863] := 16#B1D7;
   // GB2[864] := 16#B1D8;
   // GB2[865] := 16#B1D9;
   // GB2[866] := 16#B1DA;
   // GB2[867] := 16#B1DB;
   // GB2[868] := 16#B1DC;
   // GB2[869] := 16#B1DD;
   // GB2[870] := 16#B1DE;
   // GB2[871] := 16#B1DF;
   // GB2[872] := 16#B1E0;
   // GB2[873] := 16#B1E1;
   // GB2[874] := 16#B1E2;
   // GB2[875] := 16#B1E3;
   // GB2[876] := 16#B1E4;
   // GB2[877] := 16#B1E5;
   // GB2[878] := 16#B1E6;
   // GB2[879] := 16#B1E7;
   // GB2[880] := 16#B1E8;
   // GB2[881] := 16#B1E9;
   // GB2[882] := 16#B1EA;
   // GB2[883] := 16#B1EB;
   // GB2[884] := 16#B1EC;
   // GB2[885] := 16#B1ED;
   // GB2[886] := 16#B1EE;
   // GB2[887] := 16#B1EF;
   // GB2[888] := 16#B1F0;
   // GB2[889] := 16#B1F1;
   // GB2[890] := 16#B1F2;
   // GB2[891] := 16#B1F3;
   // GB2[892] := 16#B1F4;
   // GB2[893] := 16#B1F5;
   // GB2[894] := 16#B1F6;
   // GB2[895] := 16#B1F7;
   // GB2[896] := 16#B1F8;
   // GB2[897] := 16#B1F9;
   // GB2[898] := 16#B1FA;
   // GB2[899] := 16#B1FB;
   // GB2[900] := 16#B1FC;
   // GB2[901] := 16#B1FD;
   // GB2[902] := 16#B1FE;
   // GB2[903] := 16#B2A1;
   // GB2[904] := 16#B2A2;
   // GB2[905] := 16#B2A3;
   // GB2[906] := 16#B2A4;
   // GB2[907] := 16#B2A5;
   // GB2[908] := 16#B2A6;
   // GB2[909] := 16#B2A7;
   // GB2[910] := 16#B2A8;
   // GB2[911] := 16#B2A9;
   // GB2[912] := 16#B2AA;
   // GB2[913] := 16#B2AB;
   // GB2[914] := 16#B2AC;
   // GB2[915] := 16#B2AD;
   // GB2[916] := 16#B2AE;
   // GB2[917] := 16#B2AF;
   // GB2[918] := 16#B2B0;
   // GB2[919] := 16#B2B1;
   // GB2[920] := 16#B2B2;
   // GB2[921] := 16#B2B3;
   // GB2[922] := 16#B2B4;
   // GB2[923] := 16#B2B5;
   // GB2[924] := 16#B2B6;
   // GB2[925] := 16#B2B7;
   // GB2[926] := 16#B2B8;
   // GB2[927] := 16#B2B9;
   // GB2[928] := 16#B2BA;
   // GB2[929] := 16#B2BB;
   // GB2[930] := 16#B2BC;
   // GB2[931] := 16#B2BD;
   // GB2[932] := 16#B2BE;
   // GB2[933] := 16#B2BF;
   // GB2[934] := 16#B2C0;
   // GB2[935] := 16#B2C1;
   // GB2[936] := 16#B2C2;
   // GB2[937] := 16#B2C3;
   // GB2[938] := 16#B2C4;
   // GB2[939] := 16#B2C5;
   // GB2[940] := 16#B2C6;
   // GB2[941] := 16#B2C7;
   // GB2[942] := 16#B2C8;
   // GB2[943] := 16#B2C9;
   // GB2[944] := 16#B2CA;
   // GB2[945] := 16#B2CB;
   // GB2[946] := 16#B2CC;
   // GB2[947] := 16#B2CD;
   // GB2[948] := 16#B2CE;
   // GB2[949] := 16#B2CF;
   // GB2[950] := 16#B2D0;
   // GB2[951] := 16#B2D1;
   // GB2[952] := 16#B2D2;
   // GB2[953] := 16#B2D3;
   // GB2[954] := 16#B2D4;
   // GB2[955] := 16#B2D5;
   // GB2[956] := 16#B2D6;
   // GB2[957] := 16#B2D7;
   // GB2[958] := 16#B2D8;
   // GB2[959] := 16#B2D9;
   // GB2[960] := 16#B2DA;
   // GB2[961] := 16#B2DB;
   // GB2[962] := 16#B2DC;
   // GB2[963] := 16#B2DD;
   // GB2[964] := 16#B2DE;
   // GB2[965] := 16#B2DF;
   // GB2[966] := 16#B2E0;
   // GB2[967] := 16#B2E1;
   // GB2[968] := 16#B2E2;
   // GB2[969] := 16#B2E3;
   // GB2[970] := 16#B2E4;
   // GB2[971] := 16#B2E5;
   // GB2[972] := 16#B2E6;
   // GB2[973] := 16#B2E7;
   // GB2[974] := 16#B2E8;
   // GB2[975] := 16#B2E9;
   // GB2[976] := 16#B2EA;
   // GB2[977] := 16#B2EB;
   // GB2[978] := 16#B2EC;
   // GB2[979] := 16#B2ED;
   // GB2[980] := 16#B2EE;
   // GB2[981] := 16#B2EF;
   // GB2[982] := 16#B2F0;
   // GB2[983] := 16#B2F1;
   // GB2[984] := 16#B2F2;
   // GB2[985] := 16#B2F3;
   // GB2[986] := 16#B2F4;
   // GB2[987] := 16#B2F5;
   // GB2[988] := 16#B2F6;
   // GB2[989] := 16#B2F7;
   // GB2[990] := 16#B2F8;
   // GB2[991] := 16#B2F9;
   // GB2[992] := 16#B2FA;
   // GB2[993] := 16#B2FB;
   // GB2[994] := 16#B2FC;
   // GB2[995] := 16#B2FD;
   // GB2[996] := 16#B2FE;
   // GB2[997] := 16#B3A1;
   // GB2[998] := 16#B3A2;
   // GB2[999] := 16#B3A3;
   // GB2[1000] := 16#B3A4;
   // GB2[1001] := 16#B3A5;
   // GB2[1002] := 16#B3A6;
   // GB2[1003] := 16#B3A7;
   // GB2[1004] := 16#B3A8;
   // GB2[1005] := 16#B3A9;
   // GB2[1006] := 16#B3AA;
   // GB2[1007] := 16#B3AB;
   // GB2[1008] := 16#B3AC;
   // GB2[1009] := 16#B3AD;
   // GB2[1010] := 16#B3AE;
   // GB2[1011] := 16#B3AF;
   // GB2[1012] := 16#B3B0;
   // GB2[1013] := 16#B3B1;
   // GB2[1014] := 16#B3B2;
   // GB2[1015] := 16#B3B3;
   // GB2[1016] := 16#B3B4;
   // GB2[1017] := 16#B3B5;
   // GB2[1018] := 16#B3B6;
   // GB2[1019] := 16#B3B7;
   // GB2[1020] := 16#B3B8;
   // GB2[1021] := 16#B3B9;
   // GB2[1022] := 16#B3BA;
   // GB2[1023] := 16#B3BB;
   // GB2[1024] := 16#B3BC;
   // GB2[1025] := 16#B3BD;
   // GB2[1026] := 16#B3BE;
   // GB2[1027] := 16#B3BF;
   // GB2[1028] := 16#B3C0;
   // GB2[1029] := 16#B3C1;
   // GB2[1030] := 16#B3C2;
   // GB2[1031] := 16#B3C3;
   // GB2[1032] := 16#B3C4;
   // GB2[1033] := 16#B3C5;
   // GB2[1034] := 16#B3C6;
   // GB2[1035] := 16#B3C7;
   // GB2[1036] := 16#B3C8;
   // GB2[1037] := 16#B3C9;
   // GB2[1038] := 16#B3CA;
   // GB2[1039] := 16#B3CB;
   // GB2[1040] := 16#B3CC;
   // GB2[1041] := 16#B3CD;
   // GB2[1042] := 16#B3CE;
   // GB2[1043] := 16#B3CF;
   // GB2[1044] := 16#B3D0;
   // GB2[1045] := 16#B3D1;
   // GB2[1046] := 16#B3D2;
   // GB2[1047] := 16#B3D3;
   // GB2[1048] := 16#B3D4;
   // GB2[1049] := 16#B3D5;
   // GB2[1050] := 16#B3D6;
   // GB2[1051] := 16#B3D7;
   // GB2[1052] := 16#B3D8;
   // GB2[1053] := 16#B3D9;
   // GB2[1054] := 16#B3DA;
   // GB2[1055] := 16#B3DB;
   // GB2[1056] := 16#B3DC;
   // GB2[1057] := 16#B3DD;
   // GB2[1058] := 16#B3DE;
   // GB2[1059] := 16#B3DF;
   // GB2[1060] := 16#B3E0;
   // GB2[1061] := 16#B3E1;
   // GB2[1062] := 16#B3E2;
   // GB2[1063] := 16#B3E3;
   // GB2[1064] := 16#B3E4;
   // GB2[1065] := 16#B3E5;
   // GB2[1066] := 16#B3E6;
   // GB2[1067] := 16#B3E7;
   // GB2[1068] := 16#B3E8;
   // GB2[1069] := 16#B3E9;
   // GB2[1070] := 16#B3EA;
   // GB2[1071] := 16#B3EB;
   // GB2[1072] := 16#B3EC;
   // GB2[1073] := 16#B3ED;
   // GB2[1074] := 16#B3EE;
   // GB2[1075] := 16#B3EF;
   // GB2[1076] := 16#B3F0;
   // GB2[1077] := 16#B3F1;
   // GB2[1078] := 16#B3F2;
   // GB2[1079] := 16#B3F3;
   // GB2[1080] := 16#B3F4;
   // GB2[1081] := 16#B3F5;
   // GB2[1082] := 16#B3F6;
   // GB2[1083] := 16#B3F7;
   // GB2[1084] := 16#B3F8;
   // GB2[1085] := 16#B3F9;
   // GB2[1086] := 16#B3FA;
   // GB2[1087] := 16#B3FB;
   // GB2[1088] := 16#B3FC;
   // GB2[1089] := 16#B3FD;
   // GB2[1090] := 16#B3FE;
   // GB2[1091] := 16#B4A1;
   // GB2[1092] := 16#B4A2;
   // GB2[1093] := 16#B4A3;
   // GB2[1094] := 16#B4A4;
   // GB2[1095] := 16#B4A5;
   // GB2[1096] := 16#B4A6;
   // GB2[1097] := 16#B4A7;
   // GB2[1098] := 16#B4A8;
   // GB2[1099] := 16#B4A9;
   // GB2[1100] := 16#B4AA;
   // GB2[1101] := 16#B4AB;
   // GB2[1102] := 16#B4AC;
   // GB2[1103] := 16#B4AD;
   // GB2[1104] := 16#B4AE;
   // GB2[1105] := 16#B4AF;
   // GB2[1106] := 16#B4B0;
   // GB2[1107] := 16#B4B1;
   // GB2[1108] := 16#B4B2;
   // GB2[1109] := 16#B4B3;
   // GB2[1110] := 16#B4B4;
   // GB2[1111] := 16#B4B5;
   // GB2[1112] := 16#B4B6;
   // GB2[1113] := 16#B4B7;
   // GB2[1114] := 16#B4B8;
   // GB2[1115] := 16#B4B9;
   // GB2[1116] := 16#B4BA;
   // GB2[1117] := 16#B4BB;
   // GB2[1118] := 16#B4BC;
   // GB2[1119] := 16#B4BD;
   // GB2[1120] := 16#B4BE;
   // GB2[1121] := 16#B4BF;
   // GB2[1122] := 16#B4C0;
   // GB2[1123] := 16#B4C1;
   // GB2[1124] := 16#B4C2;
   // GB2[1125] := 16#B4C3;
   // GB2[1126] := 16#B4C4;
   // GB2[1127] := 16#B4C5;
   // GB2[1128] := 16#B4C6;
   // GB2[1129] := 16#B4C7;
   // GB2[1130] := 16#B4C8;
   // GB2[1131] := 16#B4C9;
   // GB2[1132] := 16#B4CA;
   // GB2[1133] := 16#B4CB;
   // GB2[1134] := 16#B4CC;
   // GB2[1135] := 16#B4CD;
   // GB2[1136] := 16#B4CE;
   // GB2[1137] := 16#B4CF;
   // GB2[1138] := 16#B4D0;
   // GB2[1139] := 16#B4D1;
   // GB2[1140] := 16#B4D2;
   // GB2[1141] := 16#B4D3;
   // GB2[1142] := 16#B4D4;
   // GB2[1143] := 16#B4D5;
   // GB2[1144] := 16#B4D6;
   // GB2[1145] := 16#B4D7;
   // GB2[1146] := 16#B4D8;
   // GB2[1147] := 16#B4D9;
   // GB2[1148] := 16#B4DA;
   // GB2[1149] := 16#B4DB;
   // GB2[1150] := 16#B4DC;
   // GB2[1151] := 16#B4DD;
   // GB2[1152] := 16#B4DE;
   // GB2[1153] := 16#B4DF;
   // GB2[1154] := 16#B4E0;
   // GB2[1155] := 16#B4E1;
   // GB2[1156] := 16#B4E2;
   // GB2[1157] := 16#B4E3;
   // GB2[1158] := 16#B4E4;
   // GB2[1159] := 16#B4E5;
   // GB2[1160] := 16#B4E6;
   // GB2[1161] := 16#B4E7;
   // GB2[1162] := 16#B4E8;
   // GB2[1163] := 16#B4E9;
   // GB2[1164] := 16#B4EA;
   // GB2[1165] := 16#B4EB;
   // GB2[1166] := 16#B4EC;
   // GB2[1167] := 16#B4ED;
   // GB2[1168] := 16#B4EE;
   // GB2[1169] := 16#B4EF;
   // GB2[1170] := 16#B4F0;
   // GB2[1171] := 16#B4F1;
   // GB2[1172] := 16#B4F2;
   // GB2[1173] := 16#B4F3;
   // GB2[1174] := 16#B4F4;
   // GB2[1175] := 16#B4F5;
   // GB2[1176] := 16#B4F6;
   // GB2[1177] := 16#B4F7;
   // GB2[1178] := 16#B4F8;
   // GB2[1179] := 16#B4F9;
   // GB2[1180] := 16#B4FA;
   // GB2[1181] := 16#B4FB;
   // GB2[1182] := 16#B4FC;
   // GB2[1183] := 16#B4FD;
   // GB2[1184] := 16#B4FE;
   // GB2[1185] := 16#B5A1;
   // GB2[1186] := 16#B5A2;
   // GB2[1187] := 16#B5A3;
   // GB2[1188] := 16#B5A4;
   // GB2[1189] := 16#B5A5;
   // GB2[1190] := 16#B5A6;
   // GB2[1191] := 16#B5A7;
   // GB2[1192] := 16#B5A8;
   // GB2[1193] := 16#B5A9;
   // GB2[1194] := 16#B5AA;
   // GB2[1195] := 16#B5AB;
   // GB2[1196] := 16#B5AC;
   // GB2[1197] := 16#B5AD;
   // GB2[1198] := 16#B5AE;
   // GB2[1199] := 16#B5AF;
   // GB2[1200] := 16#B5B0;
   // GB2[1201] := 16#B5B1;
   // GB2[1202] := 16#B5B2;
   // GB2[1203] := 16#B5B3;
   // GB2[1204] := 16#B5B4;
   // GB2[1205] := 16#B5B5;
   // GB2[1206] := 16#B5B6;
   // GB2[1207] := 16#B5B7;
   // GB2[1208] := 16#B5B8;
   // GB2[1209] := 16#B5B9;
   // GB2[1210] := 16#B5BA;
   // GB2[1211] := 16#B5BB;
   // GB2[1212] := 16#B5BC;
   // GB2[1213] := 16#B5BD;
   // GB2[1214] := 16#B5BE;
   // GB2[1215] := 16#B5BF;
   // GB2[1216] := 16#B5C0;
   // GB2[1217] := 16#B5C1;
   // GB2[1218] := 16#B5C2;
   // GB2[1219] := 16#B5C3;
   // GB2[1220] := 16#B5C4;
   // GB2[1221] := 16#B5C5;
   // GB2[1222] := 16#B5C6;
   // GB2[1223] := 16#B5C7;
   // GB2[1224] := 16#B5C8;
   // GB2[1225] := 16#B5C9;
   // GB2[1226] := 16#B5CA;
   // GB2[1227] := 16#B5CB;
   // GB2[1228] := 16#B5CC;
   // GB2[1229] := 16#B5CD;
   // GB2[1230] := 16#B5CE;
   // GB2[1231] := 16#B5CF;
   // GB2[1232] := 16#B5D0;
   // GB2[1233] := 16#B5D1;
   // GB2[1234] := 16#B5D2;
   // GB2[1235] := 16#B5D3;
   // GB2[1236] := 16#B5D4;
   // GB2[1237] := 16#B5D5;
   // GB2[1238] := 16#B5D6;
   // GB2[1239] := 16#B5D7;
   // GB2[1240] := 16#B5D8;
   // GB2[1241] := 16#B5D9;
   // GB2[1242] := 16#B5DA;
   // GB2[1243] := 16#B5DB;
   // GB2[1244] := 16#B5DC;
   // GB2[1245] := 16#B5DD;
   // GB2[1246] := 16#B5DE;
   // GB2[1247] := 16#B5DF;
   // GB2[1248] := 16#B5E0;
   // GB2[1249] := 16#B5E1;
   // GB2[1250] := 16#B5E2;
   // GB2[1251] := 16#B5E3;
   // GB2[1252] := 16#B5E4;
   // GB2[1253] := 16#B5E5;
   // GB2[1254] := 16#B5E6;
   // GB2[1255] := 16#B5E7;
   // GB2[1256] := 16#B5E8;
   // GB2[1257] := 16#B5E9;
   // GB2[1258] := 16#B5EA;
   // GB2[1259] := 16#B5EB;
   // GB2[1260] := 16#B5EC;
   // GB2[1261] := 16#B5ED;
   // GB2[1262] := 16#B5EE;
   // GB2[1263] := 16#B5EF;
   // GB2[1264] := 16#B5F0;
   // GB2[1265] := 16#B5F1;
   // GB2[1266] := 16#B5F2;
   // GB2[1267] := 16#B5F3;
   // GB2[1268] := 16#B5F4;
   // GB2[1269] := 16#B5F5;
   // GB2[1270] := 16#B5F6;
   // GB2[1271] := 16#B5F7;
   // GB2[1272] := 16#B5F8;
   // GB2[1273] := 16#B5F9;
   // GB2[1274] := 16#B5FA;
   // GB2[1275] := 16#B5FB;
   // GB2[1276] := 16#B5FC;
   // GB2[1277] := 16#B5FD;
   // GB2[1278] := 16#B5FE;
   // GB2[1279] := 16#B6A1;
   // GB2[1280] := 16#B6A2;
   // GB2[1281] := 16#B6A3;
   // GB2[1282] := 16#B6A4;
   // GB2[1283] := 16#B6A5;
   // GB2[1284] := 16#B6A6;
   // GB2[1285] := 16#B6A7;
   // GB2[1286] := 16#B6A8;
   // GB2[1287] := 16#B6A9;
   // GB2[1288] := 16#B6AA;
   // GB2[1289] := 16#B6AB;
   // GB2[1290] := 16#B6AC;
   // GB2[1291] := 16#B6AD;
   // GB2[1292] := 16#B6AE;
   // GB2[1293] := 16#B6AF;
   // GB2[1294] := 16#B6B0;
   // GB2[1295] := 16#B6B1;
   // GB2[1296] := 16#B6B2;
   // GB2[1297] := 16#B6B3;
   // GB2[1298] := 16#B6B4;
   // GB2[1299] := 16#B6B5;
   // GB2[1300] := 16#B6B6;
   // GB2[1301] := 16#B6B7;
   // GB2[1302] := 16#B6B8;
   // GB2[1303] := 16#B6B9;
   // GB2[1304] := 16#B6BA;
   // GB2[1305] := 16#B6BB;
   // GB2[1306] := 16#B6BC;
   // GB2[1307] := 16#B6BD;
   // GB2[1308] := 16#B6BE;
   // GB2[1309] := 16#B6BF;
   // GB2[1310] := 16#B6C0;
   // GB2[1311] := 16#B6C1;
   // GB2[1312] := 16#B6C2;
   // GB2[1313] := 16#B6C3;
   // GB2[1314] := 16#B6C4;
   // GB2[1315] := 16#B6C5;
   // GB2[1316] := 16#B6C6;
   // GB2[1317] := 16#B6C7;
   // GB2[1318] := 16#B6C8;
   // GB2[1319] := 16#B6C9;
   // GB2[1320] := 16#B6CA;
   // GB2[1321] := 16#B6CB;
   // GB2[1322] := 16#B6CC;
   // GB2[1323] := 16#B6CD;
   // GB2[1324] := 16#B6CE;
   // GB2[1325] := 16#B6CF;
   // GB2[1326] := 16#B6D0;
   // GB2[1327] := 16#B6D1;
   // GB2[1328] := 16#B6D2;
   // GB2[1329] := 16#B6D3;
   // GB2[1330] := 16#B6D4;
   // GB2[1331] := 16#B6D5;
   // GB2[1332] := 16#B6D6;
   // GB2[1333] := 16#B6D7;
   // GB2[1334] := 16#B6D8;
   // GB2[1335] := 16#B6D9;
   // GB2[1336] := 16#B6DA;
   // GB2[1337] := 16#B6DB;
   // GB2[1338] := 16#B6DC;
   // GB2[1339] := 16#B6DD;
   // GB2[1340] := 16#B6DE;
   // GB2[1341] := 16#B6DF;
   // GB2[1342] := 16#B6E0;
   // GB2[1343] := 16#B6E1;
   // GB2[1344] := 16#B6E2;
   // GB2[1345] := 16#B6E3;
   // GB2[1346] := 16#B6E4;
   // GB2[1347] := 16#B6E5;
   // GB2[1348] := 16#B6E6;
   // GB2[1349] := 16#B6E7;
   // GB2[1350] := 16#B6E8;
   // GB2[1351] := 16#B6E9;
   // GB2[1352] := 16#B6EA;
   // GB2[1353] := 16#B6EB;
   // GB2[1354] := 16#B6EC;
   // GB2[1355] := 16#B6ED;
   // GB2[1356] := 16#B6EE;
   // GB2[1357] := 16#B6EF;
   // GB2[1358] := 16#B6F0;
   // GB2[1359] := 16#B6F1;
   // GB2[1360] := 16#B6F2;
   // GB2[1361] := 16#B6F3;
   // GB2[1362] := 16#B6F4;
   // GB2[1363] := 16#B6F5;
   // GB2[1364] := 16#B6F6;
   // GB2[1365] := 16#B6F7;
   // GB2[1366] := 16#B6F8;
   // GB2[1367] := 16#B6F9;
   // GB2[1368] := 16#B6FA;
   // GB2[1369] := 16#B6FB;
   // GB2[1370] := 16#B6FC;
   // GB2[1371] := 16#B6FD;
   // GB2[1372] := 16#B6FE;
   // GB2[1373] := 16#B7A1;
   // GB2[1374] := 16#B7A2;
   // GB2[1375] := 16#B7A3;
   // GB2[1376] := 16#B7A4;
   // GB2[1377] := 16#B7A5;
   // GB2[1378] := 16#B7A6;
   // GB2[1379] := 16#B7A7;
   // GB2[1380] := 16#B7A8;
   // GB2[1381] := 16#B7A9;
   // GB2[1382] := 16#B7AA;
   // GB2[1383] := 16#B7AB;
   // GB2[1384] := 16#B7AC;
   // GB2[1385] := 16#B7AD;
   // GB2[1386] := 16#B7AE;
   // GB2[1387] := 16#B7AF;
   // GB2[1388] := 16#B7B0;
   // GB2[1389] := 16#B7B1;
   // GB2[1390] := 16#B7B2;
   // GB2[1391] := 16#B7B3;
   // GB2[1392] := 16#B7B4;
   // GB2[1393] := 16#B7B5;
   // GB2[1394] := 16#B7B6;
   // GB2[1395] := 16#B7B7;
   // GB2[1396] := 16#B7B8;
   // GB2[1397] := 16#B7B9;
   // GB2[1398] := 16#B7BA;
   // GB2[1399] := 16#B7BB;
   // GB2[1400] := 16#B7BC;
   // GB2[1401] := 16#B7BD;
   // GB2[1402] := 16#B7BE;
   // GB2[1403] := 16#B7BF;
   // GB2[1404] := 16#B7C0;
   // GB2[1405] := 16#B7C1;
   // GB2[1406] := 16#B7C2;
   // GB2[1407] := 16#B7C3;
   // GB2[1408] := 16#B7C4;
   // GB2[1409] := 16#B7C5;
   // GB2[1410] := 16#B7C6;
   // GB2[1411] := 16#B7C7;
   // GB2[1412] := 16#B7C8;
   // GB2[1413] := 16#B7C9;
   // GB2[1414] := 16#B7CA;
   // GB2[1415] := 16#B7CB;
   // GB2[1416] := 16#B7CC;
   // GB2[1417] := 16#B7CD;
   // GB2[1418] := 16#B7CE;
   // GB2[1419] := 16#B7CF;
   // GB2[1420] := 16#B7D0;
   // GB2[1421] := 16#B7D1;
   // GB2[1422] := 16#B7D2;
   // GB2[1423] := 16#B7D3;
   // GB2[1424] := 16#B7D4;
   // GB2[1425] := 16#B7D5;
   // GB2[1426] := 16#B7D6;
   // GB2[1427] := 16#B7D7;
   // GB2[1428] := 16#B7D8;
   // GB2[1429] := 16#B7D9;
   // GB2[1430] := 16#B7DA;
   // GB2[1431] := 16#B7DB;
   // GB2[1432] := 16#B7DC;
   // GB2[1433] := 16#B7DD;
   // GB2[1434] := 16#B7DE;
   // GB2[1435] := 16#B7DF;
   // GB2[1436] := 16#B7E0;
   // GB2[1437] := 16#B7E1;
   // GB2[1438] := 16#B7E2;
   // GB2[1439] := 16#B7E3;
   // GB2[1440] := 16#B7E4;
   // GB2[1441] := 16#B7E5;
   // GB2[1442] := 16#B7E6;
   // GB2[1443] := 16#B7E7;
   // GB2[1444] := 16#B7E8;
   // GB2[1445] := 16#B7E9;
   // GB2[1446] := 16#B7EA;
   // GB2[1447] := 16#B7EB;
   // GB2[1448] := 16#B7EC;
   // GB2[1449] := 16#B7ED;
   // GB2[1450] := 16#B7EE;
   // GB2[1451] := 16#B7EF;
   // GB2[1452] := 16#B7F0;
   // GB2[1453] := 16#B7F1;
   // GB2[1454] := 16#B7F2;
   // GB2[1455] := 16#B7F3;
   // GB2[1456] := 16#B7F4;
   // GB2[1457] := 16#B7F5;
   // GB2[1458] := 16#B7F6;
   // GB2[1459] := 16#B7F7;
   // GB2[1460] := 16#B7F8;
   // GB2[1461] := 16#B7F9;
   // GB2[1462] := 16#B7FA;
   // GB2[1463] := 16#B7FB;
   // GB2[1464] := 16#B7FC;
   // GB2[1465] := 16#B7FD;
   // GB2[1466] := 16#B7FE;
   // GB2[1467] := 16#B8A1;
   // GB2[1468] := 16#B8A2;
   // GB2[1469] := 16#B8A3;
   // GB2[1470] := 16#B8A4;
   // GB2[1471] := 16#B8A5;
   // GB2[1472] := 16#B8A6;
   // GB2[1473] := 16#B8A7;
   // GB2[1474] := 16#B8A8;
   // GB2[1475] := 16#B8A9;
   // GB2[1476] := 16#B8AA;
   // GB2[1477] := 16#B8AB;
   // GB2[1478] := 16#B8AC;
   // GB2[1479] := 16#B8AD;
   // GB2[1480] := 16#B8AE;
   // GB2[1481] := 16#B8AF;
   // GB2[1482] := 16#B8B0;
   // GB2[1483] := 16#B8B1;
   // GB2[1484] := 16#B8B2;
   // GB2[1485] := 16#B8B3;
   // GB2[1486] := 16#B8B4;
   // GB2[1487] := 16#B8B5;
   // GB2[1488] := 16#B8B6;
   // GB2[1489] := 16#B8B7;
   // GB2[1490] := 16#B8B8;
   // GB2[1491] := 16#B8B9;
   // GB2[1492] := 16#B8BA;
   // GB2[1493] := 16#B8BB;
   // GB2[1494] := 16#B8BC;
   // GB2[1495] := 16#B8BD;
   // GB2[1496] := 16#B8BE;
   // GB2[1497] := 16#B8BF;
   // GB2[1498] := 16#B8C0;
   // GB2[1499] := 16#B8C1;
   // GB2[1500] := 16#B8C2;
   // GB2[1501] := 16#B8C3;
   // GB2[1502] := 16#B8C4;
   // GB2[1503] := 16#B8C5;
   // GB2[1504] := 16#B8C6;
   // GB2[1505] := 16#B8C7;
   // GB2[1506] := 16#B8C8;
   // GB2[1507] := 16#B8C9;
   // GB2[1508] := 16#B8CA;
   // GB2[1509] := 16#B8CB;
   // GB2[1510] := 16#B8CC;
   // GB2[1511] := 16#B8CD;
   // GB2[1512] := 16#B8CE;
   // GB2[1513] := 16#B8CF;
   // GB2[1514] := 16#B8D0;
   // GB2[1515] := 16#B8D1;
   // GB2[1516] := 16#B8D2;
   // GB2[1517] := 16#B8D3;
   // GB2[1518] := 16#B8D4;
   // GB2[1519] := 16#B8D5;
   // GB2[1520] := 16#B8D6;
   // GB2[1521] := 16#B8D7;
   // GB2[1522] := 16#B8D8;
   // GB2[1523] := 16#B8D9;
   // GB2[1524] := 16#B8DA;
   // GB2[1525] := 16#B8DB;
   // GB2[1526] := 16#B8DC;
   // GB2[1527] := 16#B8DD;
   // GB2[1528] := 16#B8DE;
   // GB2[1529] := 16#B8DF;
   // GB2[1530] := 16#B8E0;
   // GB2[1531] := 16#B8E1;
   // GB2[1532] := 16#B8E2;
   // GB2[1533] := 16#B8E3;
   // GB2[1534] := 16#B8E4;
   // GB2[1535] := 16#B8E5;
   // GB2[1536] := 16#B8E6;
   // GB2[1537] := 16#B8E7;
   // GB2[1538] := 16#B8E8;
   // GB2[1539] := 16#B8E9;
   // GB2[1540] := 16#B8EA;
   // GB2[1541] := 16#B8EB;
   // GB2[1542] := 16#B8EC;
   // GB2[1543] := 16#B8ED;
   // GB2[1544] := 16#B8EE;
   // GB2[1545] := 16#B8EF;
   // GB2[1546] := 16#B8F0;
   // GB2[1547] := 16#B8F1;
   // GB2[1548] := 16#B8F2;
   // GB2[1549] := 16#B8F3;
   // GB2[1550] := 16#B8F4;
   // GB2[1551] := 16#B8F5;
   // GB2[1552] := 16#B8F6;
   // GB2[1553] := 16#B8F7;
   // GB2[1554] := 16#B8F8;
   // GB2[1555] := 16#B8F9;
   // GB2[1556] := 16#B8FA;
   // GB2[1557] := 16#B8FB;
   // GB2[1558] := 16#B8FC;
   // GB2[1559] := 16#B8FD;
   // GB2[1560] := 16#B8FE;
   // GB2[1561] := 16#B9A1;
   // GB2[1562] := 16#B9A2;
   // GB2[1563] := 16#B9A3;
   // GB2[1564] := 16#B9A4;
   // GB2[1565] := 16#B9A5;
   // GB2[1566] := 16#B9A6;
   // GB2[1567] := 16#B9A7;
   // GB2[1568] := 16#B9A8;
   // GB2[1569] := 16#B9A9;
   // GB2[1570] := 16#B9AA;
   // GB2[1571] := 16#B9AB;
   // GB2[1572] := 16#B9AC;
   // GB2[1573] := 16#B9AD;
   // GB2[1574] := 16#B9AE;
   // GB2[1575] := 16#B9AF;
   // GB2[1576] := 16#B9B0;
   // GB2[1577] := 16#B9B1;
   // GB2[1578] := 16#B9B2;
   // GB2[1579] := 16#B9B3;
   // GB2[1580] := 16#B9B4;
   // GB2[1581] := 16#B9B5;
   // GB2[1582] := 16#B9B6;
   // GB2[1583] := 16#B9B7;
   // GB2[1584] := 16#B9B8;
   // GB2[1585] := 16#B9B9;
   // GB2[1586] := 16#B9BA;
   // GB2[1587] := 16#B9BB;
   // GB2[1588] := 16#B9BC;
   // GB2[1589] := 16#B9BD;
   // GB2[1590] := 16#B9BE;
   // GB2[1591] := 16#B9BF;
   // GB2[1592] := 16#B9C0;
   // GB2[1593] := 16#B9C1;
   // GB2[1594] := 16#B9C2;
   // GB2[1595] := 16#B9C3;
   // GB2[1596] := 16#B9C4;
   // GB2[1597] := 16#B9C5;
   // GB2[1598] := 16#B9C6;
   // GB2[1599] := 16#B9C7;
   // GB2[1600] := 16#B9C8;
   // GB2[1601] := 16#B9C9;
   // GB2[1602] := 16#B9CA;
   // GB2[1603] := 16#B9CB;
   // GB2[1604] := 16#B9CC;
   // GB2[1605] := 16#B9CD;
   // GB2[1606] := 16#B9CE;
   // GB2[1607] := 16#B9CF;
   // GB2[1608] := 16#B9D0;
   // GB2[1609] := 16#B9D1;
   // GB2[1610] := 16#B9D2;
   // GB2[1611] := 16#B9D3;
   // GB2[1612] := 16#B9D4;
   // GB2[1613] := 16#B9D5;
   // GB2[1614] := 16#B9D6;
   // GB2[1615] := 16#B9D7;
   // GB2[1616] := 16#B9D8;
   // GB2[1617] := 16#B9D9;
   // GB2[1618] := 16#B9DA;
   // GB2[1619] := 16#B9DB;
   // GB2[1620] := 16#B9DC;
   // GB2[1621] := 16#B9DD;
   // GB2[1622] := 16#B9DE;
   // GB2[1623] := 16#B9DF;
   // GB2[1624] := 16#B9E0;
   // GB2[1625] := 16#B9E1;
   // GB2[1626] := 16#B9E2;
   // GB2[1627] := 16#B9E3;
   // GB2[1628] := 16#B9E4;
   // GB2[1629] := 16#B9E5;
   // GB2[1630] := 16#B9E6;
   // GB2[1631] := 16#B9E7;
   // GB2[1632] := 16#B9E8;
   // GB2[1633] := 16#B9E9;
   // GB2[1634] := 16#B9EA;
   // GB2[1635] := 16#B9EB;
   // GB2[1636] := 16#B9EC;
   // GB2[1637] := 16#B9ED;
   // GB2[1638] := 16#B9EE;
   // GB2[1639] := 16#B9EF;
   // GB2[1640] := 16#B9F0;
   // GB2[1641] := 16#B9F1;
   // GB2[1642] := 16#B9F2;
   // GB2[1643] := 16#B9F3;
   // GB2[1644] := 16#B9F4;
   // GB2[1645] := 16#B9F5;
   // GB2[1646] := 16#B9F6;
   // GB2[1647] := 16#B9F7;
   // GB2[1648] := 16#B9F8;
   // GB2[1649] := 16#B9F9;
   // GB2[1650] := 16#B9FA;
   // GB2[1651] := 16#B9FB;
   // GB2[1652] := 16#B9FC;
   // GB2[1653] := 16#B9FD;
   // GB2[1654] := 16#B9FE;
   // GB2[1655] := 16#BAA1;
   // GB2[1656] := 16#BAA2;
   // GB2[1657] := 16#BAA3;
   // GB2[1658] := 16#BAA4;
   // GB2[1659] := 16#BAA5;
   // GB2[1660] := 16#BAA6;
   // GB2[1661] := 16#BAA7;
   // GB2[1662] := 16#BAA8;
   // GB2[1663] := 16#BAA9;
   // GB2[1664] := 16#BAAA;
   // GB2[1665] := 16#BAAB;
   // GB2[1666] := 16#BAAC;
   // GB2[1667] := 16#BAAD;
   // GB2[1668] := 16#BAAE;
   // GB2[1669] := 16#BAAF;
   // GB2[1670] := 16#BAB0;
   // GB2[1671] := 16#BAB1;
   // GB2[1672] := 16#BAB2;
   // GB2[1673] := 16#BAB3;
   // GB2[1674] := 16#BAB4;
   // GB2[1675] := 16#BAB5;
   // GB2[1676] := 16#BAB6;
   // GB2[1677] := 16#BAB7;
   // GB2[1678] := 16#BAB8;
   // GB2[1679] := 16#BAB9;
   // GB2[1680] := 16#BABA;
   // GB2[1681] := 16#BABB;
   // GB2[1682] := 16#BABC;
   // GB2[1683] := 16#BABD;
   // GB2[1684] := 16#BABE;
   // GB2[1685] := 16#BABF;
   // GB2[1686] := 16#BAC0;
   // GB2[1687] := 16#BAC1;
   // GB2[1688] := 16#BAC2;
   // GB2[1689] := 16#BAC3;
   // GB2[1690] := 16#BAC4;
   // GB2[1691] := 16#BAC5;
   // GB2[1692] := 16#BAC6;
   // GB2[1693] := 16#BAC7;
   // GB2[1694] := 16#BAC8;
   // GB2[1695] := 16#BAC9;
   // GB2[1696] := 16#BACA;
   // GB2[1697] := 16#BACB;
   // GB2[1698] := 16#BACC;
   // GB2[1699] := 16#BACD;
   // GB2[1700] := 16#BACE;
   // GB2[1701] := 16#BACF;
   // GB2[1702] := 16#BAD0;
   // GB2[1703] := 16#BAD1;
   // GB2[1704] := 16#BAD2;
   // GB2[1705] := 16#BAD3;
   // GB2[1706] := 16#BAD4;
   // GB2[1707] := 16#BAD5;
   // GB2[1708] := 16#BAD6;
   // GB2[1709] := 16#BAD7;
   // GB2[1710] := 16#BAD8;
   // GB2[1711] := 16#BAD9;
   // GB2[1712] := 16#BADA;
   // GB2[1713] := 16#BADB;
   // GB2[1714] := 16#BADC;
   // GB2[1715] := 16#BADD;
   // GB2[1716] := 16#BADE;
   // GB2[1717] := 16#BADF;
   // GB2[1718] := 16#BAE0;
   // GB2[1719] := 16#BAE1;
   // GB2[1720] := 16#BAE2;
   // GB2[1721] := 16#BAE3;
   // GB2[1722] := 16#BAE4;
   // GB2[1723] := 16#BAE5;
   // GB2[1724] := 16#BAE6;
   // GB2[1725] := 16#BAE7;
   // GB2[1726] := 16#BAE8;
   // GB2[1727] := 16#BAE9;
   // GB2[1728] := 16#BAEA;
   // GB2[1729] := 16#BAEB;
   // GB2[1730] := 16#BAEC;
   // GB2[1731] := 16#BAED;
   // GB2[1732] := 16#BAEE;
   // GB2[1733] := 16#BAEF;
   // GB2[1734] := 16#BAF0;
   // GB2[1735] := 16#BAF1;
   // GB2[1736] := 16#BAF2;
   // GB2[1737] := 16#BAF3;
   // GB2[1738] := 16#BAF4;
   // GB2[1739] := 16#BAF5;
   // GB2[1740] := 16#BAF6;
   // GB2[1741] := 16#BAF7;
   // GB2[1742] := 16#BAF8;
   // GB2[1743] := 16#BAF9;
   // GB2[1744] := 16#BAFA;
   // GB2[1745] := 16#BAFB;
   // GB2[1746] := 16#BAFC;
   // GB2[1747] := 16#BAFD;
   // GB2[1748] := 16#BAFE;
   // GB2[1749] := 16#BBA1;
   // GB2[1750] := 16#BBA2;
   // GB2[1751] := 16#BBA3;
   // GB2[1752] := 16#BBA4;
   // GB2[1753] := 16#BBA5;
   // GB2[1754] := 16#BBA6;
   // GB2[1755] := 16#BBA7;
   // GB2[1756] := 16#BBA8;
   // GB2[1757] := 16#BBA9;
   // GB2[1758] := 16#BBAA;
   // GB2[1759] := 16#BBAB;
   // GB2[1760] := 16#BBAC;
   // GB2[1761] := 16#BBAD;
   // GB2[1762] := 16#BBAE;
   // GB2[1763] := 16#BBAF;
   // GB2[1764] := 16#BBB0;
   // GB2[1765] := 16#BBB1;
   // GB2[1766] := 16#BBB2;
   // GB2[1767] := 16#BBB3;
   // GB2[1768] := 16#BBB4;
   // GB2[1769] := 16#BBB5;
   // GB2[1770] := 16#BBB6;
   // GB2[1771] := 16#BBB7;
   // GB2[1772] := 16#BBB8;
   // GB2[1773] := 16#BBB9;
   // GB2[1774] := 16#BBBA;
   // GB2[1775] := 16#BBBB;
   // GB2[1776] := 16#BBBC;
   // GB2[1777] := 16#BBBD;
   // GB2[1778] := 16#BBBE;
   // GB2[1779] := 16#BBBF;
   // GB2[1780] := 16#BBC0;
   // GB2[1781] := 16#BBC1;
   // GB2[1782] := 16#BBC2;
   // GB2[1783] := 16#BBC3;
   // GB2[1784] := 16#BBC4;
   // GB2[1785] := 16#BBC5;
   // GB2[1786] := 16#BBC6;
   // GB2[1787] := 16#BBC7;
   // GB2[1788] := 16#BBC8;
   // GB2[1789] := 16#BBC9;
   // GB2[1790] := 16#BBCA;
   // GB2[1791] := 16#BBCB;
   // GB2[1792] := 16#BBCC;
   // GB2[1793] := 16#BBCD;
   // GB2[1794] := 16#BBCE;
   // GB2[1795] := 16#BBCF;
   // GB2[1796] := 16#BBD0;
   // GB2[1797] := 16#BBD1;
   // GB2[1798] := 16#BBD2;
   // GB2[1799] := 16#BBD3;
   // GB2[1800] := 16#BBD4;
   // GB2[1801] := 16#BBD5;
   // GB2[1802] := 16#BBD6;
   // GB2[1803] := 16#BBD7;
   // GB2[1804] := 16#BBD8;
   // GB2[1805] := 16#BBD9;
   // GB2[1806] := 16#BBDA;
   // GB2[1807] := 16#BBDB;
   // GB2[1808] := 16#BBDC;
   // GB2[1809] := 16#BBDD;
   // GB2[1810] := 16#BBDE;
   // GB2[1811] := 16#BBDF;
   // GB2[1812] := 16#BBE0;
   // GB2[1813] := 16#BBE1;
   // GB2[1814] := 16#BBE2;
   // GB2[1815] := 16#BBE3;
   // GB2[1816] := 16#BBE4;
   // GB2[1817] := 16#BBE5;
   // GB2[1818] := 16#BBE6;
   // GB2[1819] := 16#BBE7;
   // GB2[1820] := 16#BBE8;
   // GB2[1821] := 16#BBE9;
   // GB2[1822] := 16#BBEA;
   // GB2[1823] := 16#BBEB;
   // GB2[1824] := 16#BBEC;
   // GB2[1825] := 16#BBED;
   // GB2[1826] := 16#BBEE;
   // GB2[1827] := 16#BBEF;
   // GB2[1828] := 16#BBF0;
   // GB2[1829] := 16#BBF1;
   // GB2[1830] := 16#BBF2;
   // GB2[1831] := 16#BBF3;
   // GB2[1832] := 16#BBF4;
   // GB2[1833] := 16#BBF5;
   // GB2[1834] := 16#BBF6;
   // GB2[1835] := 16#BBF7;
   // GB2[1836] := 16#BBF8;
   // GB2[1837] := 16#BBF9;
   // GB2[1838] := 16#BBFA;
   // GB2[1839] := 16#BBFB;
   // GB2[1840] := 16#BBFC;
   // GB2[1841] := 16#BBFD;
   // GB2[1842] := 16#BBFE;
   // GB2[1843] := 16#BCA1;
   // GB2[1844] := 16#BCA2;
   // GB2[1845] := 16#BCA3;
   // GB2[1846] := 16#BCA4;
   // GB2[1847] := 16#BCA5;
   // GB2[1848] := 16#BCA6;
   // GB2[1849] := 16#BCA7;
   // GB2[1850] := 16#BCA8;
   // GB2[1851] := 16#BCA9;
   // GB2[1852] := 16#BCAA;
   // GB2[1853] := 16#BCAB;
   // GB2[1854] := 16#BCAC;
   // GB2[1855] := 16#BCAD;
   // GB2[1856] := 16#BCAE;
   // GB2[1857] := 16#BCAF;
   // GB2[1858] := 16#BCB0;
   // GB2[1859] := 16#BCB1;
   // GB2[1860] := 16#BCB2;
   // GB2[1861] := 16#BCB3;
   // GB2[1862] := 16#BCB4;
   // GB2[1863] := 16#BCB5;
   // GB2[1864] := 16#BCB6;
   // GB2[1865] := 16#BCB7;
   // GB2[1866] := 16#BCB8;
   // GB2[1867] := 16#BCB9;
   // GB2[1868] := 16#BCBA;
   // GB2[1869] := 16#BCBB;
   // GB2[1870] := 16#BCBC;
   // GB2[1871] := 16#BCBD;
   // GB2[1872] := 16#BCBE;
   // GB2[1873] := 16#BCBF;
   // GB2[1874] := 16#BCC0;
   // GB2[1875] := 16#BCC1;
   // GB2[1876] := 16#BCC2;
   // GB2[1877] := 16#BCC3;
   // GB2[1878] := 16#BCC4;
   // GB2[1879] := 16#BCC5;
   // GB2[1880] := 16#BCC6;
   // GB2[1881] := 16#BCC7;
   // GB2[1882] := 16#BCC8;
   // GB2[1883] := 16#BCC9;
   // GB2[1884] := 16#BCCA;
   // GB2[1885] := 16#BCCB;
   // GB2[1886] := 16#BCCC;
   // GB2[1887] := 16#BCCD;
   // GB2[1888] := 16#BCCE;
   // GB2[1889] := 16#BCCF;
   // GB2[1890] := 16#BCD0;
   // GB2[1891] := 16#BCD1;
   // GB2[1892] := 16#BCD2;
   // GB2[1893] := 16#BCD3;
   // GB2[1894] := 16#BCD4;
   // GB2[1895] := 16#BCD5;
   // GB2[1896] := 16#BCD6;
   // GB2[1897] := 16#BCD7;
   // GB2[1898] := 16#BCD8;
   // GB2[1899] := 16#BCD9;
   // GB2[1900] := 16#BCDA;
   // GB2[1901] := 16#BCDB;
   // GB2[1902] := 16#BCDC;
   // GB2[1903] := 16#BCDD;
   // GB2[1904] := 16#BCDE;
   // GB2[1905] := 16#BCDF;
   // GB2[1906] := 16#BCE0;
   // GB2[1907] := 16#BCE1;
   // GB2[1908] := 16#BCE2;
   // GB2[1909] := 16#BCE3;
   // GB2[1910] := 16#BCE4;
   // GB2[1911] := 16#BCE5;
   // GB2[1912] := 16#BCE6;
   // GB2[1913] := 16#BCE7;
   // GB2[1914] := 16#BCE8;
   // GB2[1915] := 16#BCE9;
   // GB2[1916] := 16#BCEA;
   // GB2[1917] := 16#BCEB;
   // GB2[1918] := 16#BCEC;
   // GB2[1919] := 16#BCED;
   // GB2[1920] := 16#BCEE;
   // GB2[1921] := 16#BCEF;
   // GB2[1922] := 16#BCF0;
   // GB2[1923] := 16#BCF1;
   // GB2[1924] := 16#BCF2;
   // GB2[1925] := 16#BCF3;
   // GB2[1926] := 16#BCF4;
   // GB2[1927] := 16#BCF5;
   // GB2[1928] := 16#BCF6;
   // GB2[1929] := 16#BCF7;
   // GB2[1930] := 16#BCF8;
   // GB2[1931] := 16#BCF9;
   // GB2[1932] := 16#BCFA;
   // GB2[1933] := 16#BCFB;
   // GB2[1934] := 16#BCFC;
   // GB2[1935] := 16#BCFD;
   // GB2[1936] := 16#BCFE;
   // GB2[1937] := 16#BDA1;
   // GB2[1938] := 16#BDA2;
   // GB2[1939] := 16#BDA3;
   // GB2[1940] := 16#BDA4;
   // GB2[1941] := 16#BDA5;
   // GB2[1942] := 16#BDA6;
   // GB2[1943] := 16#BDA7;
   // GB2[1944] := 16#BDA8;
   // GB2[1945] := 16#BDA9;
   // GB2[1946] := 16#BDAA;
   // GB2[1947] := 16#BDAB;
   // GB2[1948] := 16#BDAC;
   // GB2[1949] := 16#BDAD;
   // GB2[1950] := 16#BDAE;
   // GB2[1951] := 16#BDAF;
   // GB2[1952] := 16#BDB0;
   // GB2[1953] := 16#BDB1;
   // GB2[1954] := 16#BDB2;
   // GB2[1955] := 16#BDB3;
   // GB2[1956] := 16#BDB4;
   // GB2[1957] := 16#BDB5;
   // GB2[1958] := 16#BDB6;
   // GB2[1959] := 16#BDB7;
   // GB2[1960] := 16#BDB8;
   // GB2[1961] := 16#BDB9;
   // GB2[1962] := 16#BDBA;
   // GB2[1963] := 16#BDBB;
   // GB2[1964] := 16#BDBC;
   // GB2[1965] := 16#BDBD;
   // GB2[1966] := 16#BDBE;
   // GB2[1967] := 16#BDBF;
   // GB2[1968] := 16#BDC0;
   // GB2[1969] := 16#BDC1;
   // GB2[1970] := 16#BDC2;
   // GB2[1971] := 16#BDC3;
   // GB2[1972] := 16#BDC4;
   // GB2[1973] := 16#BDC5;
   // GB2[1974] := 16#BDC6;
   // GB2[1975] := 16#BDC7;
   // GB2[1976] := 16#BDC8;
   // GB2[1977] := 16#BDC9;
   // GB2[1978] := 16#BDCA;
   // GB2[1979] := 16#BDCB;
   // GB2[1980] := 16#BDCC;
   // GB2[1981] := 16#BDCD;
   // GB2[1982] := 16#BDCE;
   // GB2[1983] := 16#BDCF;
   // GB2[1984] := 16#BDD0;
   // GB2[1985] := 16#BDD1;
   // GB2[1986] := 16#BDD2;
   // GB2[1987] := 16#BDD3;
   // GB2[1988] := 16#BDD4;
   // GB2[1989] := 16#BDD5;
   // GB2[1990] := 16#BDD6;
   // GB2[1991] := 16#BDD7;
   // GB2[1992] := 16#BDD8;
   // GB2[1993] := 16#BDD9;
   // GB2[1994] := 16#BDDA;
   // GB2[1995] := 16#BDDB;
   // GB2[1996] := 16#BDDC;
   // GB2[1997] := 16#BDDD;
   // GB2[1998] := 16#BDDE;
   // GB2[1999] := 16#BDDF;
   // GB2[2000] := 16#BDE0;
   // GB2[2001] := 16#BDE1;
   // GB2[2002] := 16#BDE2;
   // GB2[2003] := 16#BDE3;
   // GB2[2004] := 16#BDE4;
   // GB2[2005] := 16#BDE5;
   // GB2[2006] := 16#BDE6;
   // GB2[2007] := 16#BDE7;
   // GB2[2008] := 16#BDE8;
   // GB2[2009] := 16#BDE9;
   // GB2[2010] := 16#BDEA;
   // GB2[2011] := 16#BDEB;
   // GB2[2012] := 16#BDEC;
   // GB2[2013] := 16#BDED;
   // GB2[2014] := 16#BDEE;
   // GB2[2015] := 16#BDEF;
   // GB2[2016] := 16#BDF0;
   // GB2[2017] := 16#BDF1;
   // GB2[2018] := 16#BDF2;
   // GB2[2019] := 16#BDF3;
   // GB2[2020] := 16#BDF4;
   // GB2[2021] := 16#BDF5;
   // GB2[2022] := 16#BDF6;
   // GB2[2023] := 16#BDF7;
   // GB2[2024] := 16#BDF8;
   // GB2[2025] := 16#BDF9;
   // GB2[2026] := 16#BDFA;
   // GB2[2027] := 16#BDFB;
   // GB2[2028] := 16#BDFC;
   // GB2[2029] := 16#BDFD;
   // GB2[2030] := 16#BDFE;
   // GB2[2031] := 16#BEA1;
   // GB2[2032] := 16#BEA2;
   // GB2[2033] := 16#BEA3;
   // GB2[2034] := 16#BEA4;
   // GB2[2035] := 16#BEA5;
   // GB2[2036] := 16#BEA6;
   // GB2[2037] := 16#BEA7;
   // GB2[2038] := 16#BEA8;
   // GB2[2039] := 16#BEA9;
   // GB2[2040] := 16#BEAA;
   // GB2[2041] := 16#BEAB;
   // GB2[2042] := 16#BEAC;
   // GB2[2043] := 16#BEAD;
   // GB2[2044] := 16#BEAE;
   // GB2[2045] := 16#BEAF;
   // GB2[2046] := 16#BEB0;
   // GB2[2047] := 16#BEB1;
   // GB2[2048] := 16#BEB2;
   // GB2[2049] := 16#BEB3;
   // GB2[2050] := 16#BEB4;
   // GB2[2051] := 16#BEB5;
   // GB2[2052] := 16#BEB6;
   // GB2[2053] := 16#BEB7;
   // GB2[2054] := 16#BEB8;
   // GB2[2055] := 16#BEB9;
   // GB2[2056] := 16#BEBA;
   // GB2[2057] := 16#BEBB;
   // GB2[2058] := 16#BEBC;
   // GB2[2059] := 16#BEBD;
   // GB2[2060] := 16#BEBE;
   // GB2[2061] := 16#BEBF;
   // GB2[2062] := 16#BEC0;
   // GB2[2063] := 16#BEC1;
   // GB2[2064] := 16#BEC2;
   // GB2[2065] := 16#BEC3;
   // GB2[2066] := 16#BEC4;
   // GB2[2067] := 16#BEC5;
   // GB2[2068] := 16#BEC6;
   // GB2[2069] := 16#BEC7;
   // GB2[2070] := 16#BEC8;
   // GB2[2071] := 16#BEC9;
   // GB2[2072] := 16#BECA;
   // GB2[2073] := 16#BECB;
   // GB2[2074] := 16#BECC;
   // GB2[2075] := 16#BECD;
   // GB2[2076] := 16#BECE;
   // GB2[2077] := 16#BECF;
   // GB2[2078] := 16#BED0;
   // GB2[2079] := 16#BED1;
   // GB2[2080] := 16#BED2;
   // GB2[2081] := 16#BED3;
   // GB2[2082] := 16#BED4;
   // GB2[2083] := 16#BED5;
   // GB2[2084] := 16#BED6;
   // GB2[2085] := 16#BED7;
   // GB2[2086] := 16#BED8;
   // GB2[2087] := 16#BED9;
   // GB2[2088] := 16#BEDA;
   // GB2[2089] := 16#BEDB;
   // GB2[2090] := 16#BEDC;
   // GB2[2091] := 16#BEDD;
   // GB2[2092] := 16#BEDE;
   // GB2[2093] := 16#BEDF;
   // GB2[2094] := 16#BEE0;
   // GB2[2095] := 16#BEE1;
   // GB2[2096] := 16#BEE2;
   // GB2[2097] := 16#BEE3;
   // GB2[2098] := 16#BEE4;
   // GB2[2099] := 16#BEE5;
   // GB2[2100] := 16#BEE6;
   // GB2[2101] := 16#BEE7;
   // GB2[2102] := 16#BEE8;
   // GB2[2103] := 16#BEE9;
   // GB2[2104] := 16#BEEA;
   // GB2[2105] := 16#BEEB;
   // GB2[2106] := 16#BEEC;
   // GB2[2107] := 16#BEED;
   // GB2[2108] := 16#BEEE;
   // GB2[2109] := 16#BEEF;
   // GB2[2110] := 16#BEF0;
   // GB2[2111] := 16#BEF1;
   // GB2[2112] := 16#BEF2;
   // GB2[2113] := 16#BEF3;
   // GB2[2114] := 16#BEF4;
   // GB2[2115] := 16#BEF5;
   // GB2[2116] := 16#BEF6;
   // GB2[2117] := 16#BEF7;
   // GB2[2118] := 16#BEF8;
   // GB2[2119] := 16#BEF9;
   // GB2[2120] := 16#BEFA;
   // GB2[2121] := 16#BEFB;
   // GB2[2122] := 16#BEFC;
   // GB2[2123] := 16#BEFD;
   // GB2[2124] := 16#BEFE;
   // GB2[2125] := 16#BFA1;
   // GB2[2126] := 16#BFA2;
   // GB2[2127] := 16#BFA3;
   // GB2[2128] := 16#BFA4;
   // GB2[2129] := 16#BFA5;
   // GB2[2130] := 16#BFA6;
   // GB2[2131] := 16#BFA7;
   // GB2[2132] := 16#BFA8;
   // GB2[2133] := 16#BFA9;
   // GB2[2134] := 16#BFAA;
   // GB2[2135] := 16#BFAB;
   // GB2[2136] := 16#BFAC;
   // GB2[2137] := 16#BFAD;
   // GB2[2138] := 16#BFAE;
   // GB2[2139] := 16#BFAF;
   // GB2[2140] := 16#BFB0;
   // GB2[2141] := 16#BFB1;
   // GB2[2142] := 16#BFB2;
   // GB2[2143] := 16#BFB3;
   // GB2[2144] := 16#BFB4;
   // GB2[2145] := 16#BFB5;
   // GB2[2146] := 16#BFB6;
   // GB2[2147] := 16#BFB7;
   // GB2[2148] := 16#BFB8;
   // GB2[2149] := 16#BFB9;
   // GB2[2150] := 16#BFBA;
   // GB2[2151] := 16#BFBB;
   // GB2[2152] := 16#BFBC;
   // GB2[2153] := 16#BFBD;
   // GB2[2154] := 16#BFBE;
   // GB2[2155] := 16#BFBF;
   // GB2[2156] := 16#BFC0;
   // GB2[2157] := 16#BFC1;
   // GB2[2158] := 16#BFC2;
   // GB2[2159] := 16#BFC3;
   // GB2[2160] := 16#BFC4;
   // GB2[2161] := 16#BFC5;
   // GB2[2162] := 16#BFC6;
   // GB2[2163] := 16#BFC7;
   // GB2[2164] := 16#BFC8;
   // GB2[2165] := 16#BFC9;
   // GB2[2166] := 16#BFCA;
   // GB2[2167] := 16#BFCB;
   // GB2[2168] := 16#BFCC;
   // GB2[2169] := 16#BFCD;
   // GB2[2170] := 16#BFCE;
   // GB2[2171] := 16#BFCF;
   // GB2[2172] := 16#BFD0;
   // GB2[2173] := 16#BFD1;
   // GB2[2174] := 16#BFD2;
   // GB2[2175] := 16#BFD3;
   // GB2[2176] := 16#BFD4;
   // GB2[2177] := 16#BFD5;
   // GB2[2178] := 16#BFD6;
   // GB2[2179] := 16#BFD7;
   // GB2[2180] := 16#BFD8;
   // GB2[2181] := 16#BFD9;
   // GB2[2182] := 16#BFDA;
   // GB2[2183] := 16#BFDB;
   // GB2[2184] := 16#BFDC;
   // GB2[2185] := 16#BFDD;
   // GB2[2186] := 16#BFDE;
   // GB2[2187] := 16#BFDF;
   // GB2[2188] := 16#BFE0;
   // GB2[2189] := 16#BFE1;
   // GB2[2190] := 16#BFE2;
   // GB2[2191] := 16#BFE3;
   // GB2[2192] := 16#BFE4;
   // GB2[2193] := 16#BFE5;
   // GB2[2194] := 16#BFE6;
   // GB2[2195] := 16#BFE7;
   // GB2[2196] := 16#BFE8;
   // GB2[2197] := 16#BFE9;
   // GB2[2198] := 16#BFEA;
   // GB2[2199] := 16#BFEB;
   // GB2[2200] := 16#BFEC;
   // GB2[2201] := 16#BFED;
   // GB2[2202] := 16#BFEE;
   // GB2[2203] := 16#BFEF;
   // GB2[2204] := 16#BFF0;
   // GB2[2205] := 16#BFF1;
   // GB2[2206] := 16#BFF2;
   // GB2[2207] := 16#BFF3;
   // GB2[2208] := 16#BFF4;
   // GB2[2209] := 16#BFF5;
   // GB2[2210] := 16#BFF6;
   // GB2[2211] := 16#BFF7;
   // GB2[2212] := 16#BFF8;
   // GB2[2213] := 16#BFF9;
   // GB2[2214] := 16#BFFA;
   // GB2[2215] := 16#BFFB;
   // GB2[2216] := 16#BFFC;
   // GB2[2217] := 16#BFFD;
   // GB2[2218] := 16#BFFE;
   // GB2[2219] := 16#C0A1;
   // GB2[2220] := 16#C0A2;
   // GB2[2221] := 16#C0A3;
   // GB2[2222] := 16#C0A4;
   // GB2[2223] := 16#C0A5;
   // GB2[2224] := 16#C0A6;
   // GB2[2225] := 16#C0A7;
   // GB2[2226] := 16#C0A8;
   // GB2[2227] := 16#C0A9;
   // GB2[2228] := 16#C0AA;
   // GB2[2229] := 16#C0AB;
   // GB2[2230] := 16#C0AC;
   // GB2[2231] := 16#C0AD;
   // GB2[2232] := 16#C0AE;
   // GB2[2233] := 16#C0AF;
   // GB2[2234] := 16#C0B0;
   // GB2[2235] := 16#C0B1;
   // GB2[2236] := 16#C0B2;
   // GB2[2237] := 16#C0B3;
   // GB2[2238] := 16#C0B4;
   // GB2[2239] := 16#C0B5;
   // GB2[2240] := 16#C0B6;
   // GB2[2241] := 16#C0B7;
   // GB2[2242] := 16#C0B8;
   // GB2[2243] := 16#C0B9;
   // GB2[2244] := 16#C0BA;
   // GB2[2245] := 16#C0BB;
   // GB2[2246] := 16#C0BC;
   // GB2[2247] := 16#C0BD;
   // GB2[2248] := 16#C0BE;
   // GB2[2249] := 16#C0BF;
   // GB2[2250] := 16#C0C0;
   // GB2[2251] := 16#C0C1;
   // GB2[2252] := 16#C0C2;
   // GB2[2253] := 16#C0C3;
   // GB2[2254] := 16#C0C4;
   // GB2[2255] := 16#C0C5;
   // GB2[2256] := 16#C0C6;
   // GB2[2257] := 16#C0C7;
   // GB2[2258] := 16#C0C8;
   // GB2[2259] := 16#C0C9;
   // GB2[2260] := 16#C0CA;
   // GB2[2261] := 16#C0CB;
   // GB2[2262] := 16#C0CC;
   // GB2[2263] := 16#C0CD;
   // GB2[2264] := 16#C0CE;
   // GB2[2265] := 16#C0CF;
   // GB2[2266] := 16#C0D0;
   // GB2[2267] := 16#C0D1;
   // GB2[2268] := 16#C0D2;
   // GB2[2269] := 16#C0D3;
   // GB2[2270] := 16#C0D4;
   // GB2[2271] := 16#C0D5;
   // GB2[2272] := 16#C0D6;
   // GB2[2273] := 16#C0D7;
   // GB2[2274] := 16#C0D8;
   // GB2[2275] := 16#C0D9;
   // GB2[2276] := 16#C0DA;
   // GB2[2277] := 16#C0DB;
   // GB2[2278] := 16#C0DC;
   // GB2[2279] := 16#C0DD;
   // GB2[2280] := 16#C0DE;
   // GB2[2281] := 16#C0DF;
   // GB2[2282] := 16#C0E0;
   // GB2[2283] := 16#C0E1;
   // GB2[2284] := 16#C0E2;
   // GB2[2285] := 16#C0E3;
   // GB2[2286] := 16#C0E4;
   // GB2[2287] := 16#C0E5;
   // GB2[2288] := 16#C0E6;
   // GB2[2289] := 16#C0E7;
   // GB2[2290] := 16#C0E8;
   // GB2[2291] := 16#C0E9;
   // GB2[2292] := 16#C0EA;
   // GB2[2293] := 16#C0EB;
   // GB2[2294] := 16#C0EC;
   // GB2[2295] := 16#C0ED;
   // GB2[2296] := 16#C0EE;
   // GB2[2297] := 16#C0EF;
   // GB2[2298] := 16#C0F0;
   // GB2[2299] := 16#C0F1;
   // GB2[2300] := 16#C0F2;
   // GB2[2301] := 16#C0F3;
   // GB2[2302] := 16#C0F4;
   // GB2[2303] := 16#C0F5;
   // GB2[2304] := 16#C0F6;
   // GB2[2305] := 16#C0F7;
   // GB2[2306] := 16#C0F8;
   // GB2[2307] := 16#C0F9;
   // GB2[2308] := 16#C0FA;
   // GB2[2309] := 16#C0FB;
   // GB2[2310] := 16#C0FC;
   // GB2[2311] := 16#C0FD;
   // GB2[2312] := 16#C0FE;
   // GB2[2313] := 16#C1A1;
   // GB2[2314] := 16#C1A2;
   // GB2[2315] := 16#C1A3;
   // GB2[2316] := 16#C1A4;
   // GB2[2317] := 16#C1A5;
   // GB2[2318] := 16#C1A6;
   // GB2[2319] := 16#C1A7;
   // GB2[2320] := 16#C1A8;
   // GB2[2321] := 16#C1A9;
   // GB2[2322] := 16#C1AA;
   // GB2[2323] := 16#C1AB;
   // GB2[2324] := 16#C1AC;
   // GB2[2325] := 16#C1AD;
   // GB2[2326] := 16#C1AE;
   // GB2[2327] := 16#C1AF;
   // GB2[2328] := 16#C1B0;
   // GB2[2329] := 16#C1B1;
   // GB2[2330] := 16#C1B2;
   // GB2[2331] := 16#C1B3;
   // GB2[2332] := 16#C1B4;
   // GB2[2333] := 16#C1B5;
   // GB2[2334] := 16#C1B6;
   // GB2[2335] := 16#C1B7;
   // GB2[2336] := 16#C1B8;
   // GB2[2337] := 16#C1B9;
   // GB2[2338] := 16#C1BA;
   // GB2[2339] := 16#C1BB;
   // GB2[2340] := 16#C1BC;
   // GB2[2341] := 16#C1BD;
   // GB2[2342] := 16#C1BE;
   // GB2[2343] := 16#C1BF;
   // GB2[2344] := 16#C1C0;
   // GB2[2345] := 16#C1C1;
   // GB2[2346] := 16#C1C2;
   // GB2[2347] := 16#C1C3;
   // GB2[2348] := 16#C1C4;
   // GB2[2349] := 16#C1C5;
   // GB2[2350] := 16#C1C6;
   // GB2[2351] := 16#C1C7;
   // GB2[2352] := 16#C1C8;
   // GB2[2353] := 16#C1C9;
   // GB2[2354] := 16#C1CA;
   // GB2[2355] := 16#C1CB;
   // GB2[2356] := 16#C1CC;
   // GB2[2357] := 16#C1CD;
   // GB2[2358] := 16#C1CE;
   // GB2[2359] := 16#C1CF;
   // GB2[2360] := 16#C1D0;
   // GB2[2361] := 16#C1D1;
   // GB2[2362] := 16#C1D2;
   // GB2[2363] := 16#C1D3;
   // GB2[2364] := 16#C1D4;
   // GB2[2365] := 16#C1D5;
   // GB2[2366] := 16#C1D6;
   // GB2[2367] := 16#C1D7;
   // GB2[2368] := 16#C1D8;
   // GB2[2369] := 16#C1D9;
   // GB2[2370] := 16#C1DA;
   // GB2[2371] := 16#C1DB;
   // GB2[2372] := 16#C1DC;
   // GB2[2373] := 16#C1DD;
   // GB2[2374] := 16#C1DE;
   // GB2[2375] := 16#C1DF;
   // GB2[2376] := 16#C1E0;
   // GB2[2377] := 16#C1E1;
   // GB2[2378] := 16#C1E2;
   // GB2[2379] := 16#C1E3;
   // GB2[2380] := 16#C1E4;
   // GB2[2381] := 16#C1E5;
   // GB2[2382] := 16#C1E6;
   // GB2[2383] := 16#C1E7;
   // GB2[2384] := 16#C1E8;
   // GB2[2385] := 16#C1E9;
   // GB2[2386] := 16#C1EA;
   // GB2[2387] := 16#C1EB;
   // GB2[2388] := 16#C1EC;
   // GB2[2389] := 16#C1ED;
   // GB2[2390] := 16#C1EE;
   // GB2[2391] := 16#C1EF;
   // GB2[2392] := 16#C1F0;
   // GB2[2393] := 16#C1F1;
   // GB2[2394] := 16#C1F2;
   // GB2[2395] := 16#C1F3;
   // GB2[2396] := 16#C1F4;
   // GB2[2397] := 16#C1F5;
   // GB2[2398] := 16#C1F6;
   // GB2[2399] := 16#C1F7;
   // GB2[2400] := 16#C1F8;
   // GB2[2401] := 16#C1F9;
   // GB2[2402] := 16#C1FA;
   // GB2[2403] := 16#C1FB;
   // GB2[2404] := 16#C1FC;
   // GB2[2405] := 16#C1FD;
   // GB2[2406] := 16#C1FE;
   // GB2[2407] := 16#C2A1;
   // GB2[2408] := 16#C2A2;
   // GB2[2409] := 16#C2A3;
   // GB2[2410] := 16#C2A4;
   // GB2[2411] := 16#C2A5;
   // GB2[2412] := 16#C2A6;
   // GB2[2413] := 16#C2A7;
   // GB2[2414] := 16#C2A8;
   // GB2[2415] := 16#C2A9;
   // GB2[2416] := 16#C2AA;
   // GB2[2417] := 16#C2AB;
   // GB2[2418] := 16#C2AC;
   // GB2[2419] := 16#C2AD;
   // GB2[2420] := 16#C2AE;
   // GB2[2421] := 16#C2AF;
   // GB2[2422] := 16#C2B0;
   // GB2[2423] := 16#C2B1;
   // GB2[2424] := 16#C2B2;
   // GB2[2425] := 16#C2B3;
   // GB2[2426] := 16#C2B4;
   // GB2[2427] := 16#C2B5;
   // GB2[2428] := 16#C2B6;
   // GB2[2429] := 16#C2B7;
   // GB2[2430] := 16#C2B8;
   // GB2[2431] := 16#C2B9;
   // GB2[2432] := 16#C2BA;
   // GB2[2433] := 16#C2BB;
   // GB2[2434] := 16#C2BC;
   // GB2[2435] := 16#C2BD;
   // GB2[2436] := 16#C2BE;
   // GB2[2437] := 16#C2BF;
   // GB2[2438] := 16#C2C0;
   // GB2[2439] := 16#C2C1;
   // GB2[2440] := 16#C2C2;
   // GB2[2441] := 16#C2C3;
   // GB2[2442] := 16#C2C4;
   // GB2[2443] := 16#C2C5;
   // GB2[2444] := 16#C2C6;
   // GB2[2445] := 16#C2C7;
   // GB2[2446] := 16#C2C8;
   // GB2[2447] := 16#C2C9;
   // GB2[2448] := 16#C2CA;
   // GB2[2449] := 16#C2CB;
   // GB2[2450] := 16#C2CC;
   // GB2[2451] := 16#C2CD;
   // GB2[2452] := 16#C2CE;
   // GB2[2453] := 16#C2CF;
   // GB2[2454] := 16#C2D0;
   // GB2[2455] := 16#C2D1;
   // GB2[2456] := 16#C2D2;
   // GB2[2457] := 16#C2D3;
   // GB2[2458] := 16#C2D4;
   // GB2[2459] := 16#C2D5;
   // GB2[2460] := 16#C2D6;
   // GB2[2461] := 16#C2D7;
   // GB2[2462] := 16#C2D8;
   // GB2[2463] := 16#C2D9;
   // GB2[2464] := 16#C2DA;
   // GB2[2465] := 16#C2DB;
   // GB2[2466] := 16#C2DC;
   // GB2[2467] := 16#C2DD;
   // GB2[2468] := 16#C2DE;
   // GB2[2469] := 16#C2DF;
   // GB2[2470] := 16#C2E0;
   // GB2[2471] := 16#C2E1;
   // GB2[2472] := 16#C2E2;
   // GB2[2473] := 16#C2E3;
   // GB2[2474] := 16#C2E4;
   // GB2[2475] := 16#C2E5;
   // GB2[2476] := 16#C2E6;
   // GB2[2477] := 16#C2E7;
   // GB2[2478] := 16#C2E8;
   // GB2[2479] := 16#C2E9;
   // GB2[2480] := 16#C2EA;
   // GB2[2481] := 16#C2EB;
   // GB2[2482] := 16#C2EC;
   // GB2[2483] := 16#C2ED;
   // GB2[2484] := 16#C2EE;
   // GB2[2485] := 16#C2EF;
   // GB2[2486] := 16#C2F0;
   // GB2[2487] := 16#C2F1;
   // GB2[2488] := 16#C2F2;
   // GB2[2489] := 16#C2F3;
   // GB2[2490] := 16#C2F4;
   // GB2[2491] := 16#C2F5;
   // GB2[2492] := 16#C2F6;
   // GB2[2493] := 16#C2F7;
   // GB2[2494] := 16#C2F8;
   // GB2[2495] := 16#C2F9;
   // GB2[2496] := 16#C2FA;
   // GB2[2497] := 16#C2FB;
   // GB2[2498] := 16#C2FC;
   // GB2[2499] := 16#C2FD;
   // GB2[2500] := 16#C2FE;
   // GB2[2501] := 16#C3A1;
   // GB2[2502] := 16#C3A2;
   // GB2[2503] := 16#C3A3;
   // GB2[2504] := 16#C3A4;
   // GB2[2505] := 16#C3A5;
   // GB2[2506] := 16#C3A6;
   // GB2[2507] := 16#C3A7;
   // GB2[2508] := 16#C3A8;
   // GB2[2509] := 16#C3A9;
   // GB2[2510] := 16#C3AA;
   // GB2[2511] := 16#C3AB;
   // GB2[2512] := 16#C3AC;
   // GB2[2513] := 16#C3AD;
   // GB2[2514] := 16#C3AE;
   // GB2[2515] := 16#C3AF;
   // GB2[2516] := 16#C3B0;
   // GB2[2517] := 16#C3B1;
   // GB2[2518] := 16#C3B2;
   // GB2[2519] := 16#C3B3;
   // GB2[2520] := 16#C3B4;
   // GB2[2521] := 16#C3B5;
   // GB2[2522] := 16#C3B6;
   // GB2[2523] := 16#C3B7;
   // GB2[2524] := 16#C3B8;
   // GB2[2525] := 16#C3B9;
   // GB2[2526] := 16#C3BA;
   // GB2[2527] := 16#C3BB;
   // GB2[2528] := 16#C3BC;
   // GB2[2529] := 16#C3BD;
   // GB2[2530] := 16#C3BE;
   // GB2[2531] := 16#C3BF;
   // GB2[2532] := 16#C3C0;
   // GB2[2533] := 16#C3C1;
   // GB2[2534] := 16#C3C2;
   // GB2[2535] := 16#C3C3;
   // GB2[2536] := 16#C3C4;
   // GB2[2537] := 16#C3C5;
   // GB2[2538] := 16#C3C6;
   // GB2[2539] := 16#C3C7;
   // GB2[2540] := 16#C3C8;
   // GB2[2541] := 16#C3C9;
   // GB2[2542] := 16#C3CA;
   // GB2[2543] := 16#C3CB;
   // GB2[2544] := 16#C3CC;
   // GB2[2545] := 16#C3CD;
   // GB2[2546] := 16#C3CE;
   // GB2[2547] := 16#C3CF;
   // GB2[2548] := 16#C3D0;
   // GB2[2549] := 16#C3D1;
   // GB2[2550] := 16#C3D2;
   // GB2[2551] := 16#C3D3;
   // GB2[2552] := 16#C3D4;
   // GB2[2553] := 16#C3D5;
   // GB2[2554] := 16#C3D6;
   // GB2[2555] := 16#C3D7;
   // GB2[2556] := 16#C3D8;
   // GB2[2557] := 16#C3D9;
   // GB2[2558] := 16#C3DA;
   // GB2[2559] := 16#C3DB;
   // GB2[2560] := 16#C3DC;
   // GB2[2561] := 16#C3DD;
   // GB2[2562] := 16#C3DE;
   // GB2[2563] := 16#C3DF;
   // GB2[2564] := 16#C3E0;
   // GB2[2565] := 16#C3E1;
   // GB2[2566] := 16#C3E2;
   // GB2[2567] := 16#C3E3;
   // GB2[2568] := 16#C3E4;
   // GB2[2569] := 16#C3E5;
   // GB2[2570] := 16#C3E6;
   // GB2[2571] := 16#C3E7;
   // GB2[2572] := 16#C3E8;
   // GB2[2573] := 16#C3E9;
   // GB2[2574] := 16#C3EA;
   // GB2[2575] := 16#C3EB;
   // GB2[2576] := 16#C3EC;
   // GB2[2577] := 16#C3ED;
   // GB2[2578] := 16#C3EE;
   // GB2[2579] := 16#C3EF;
   // GB2[2580] := 16#C3F0;
   // GB2[2581] := 16#C3F1;
   // GB2[2582] := 16#C3F2;
   // GB2[2583] := 16#C3F3;
   // GB2[2584] := 16#C3F4;
   // GB2[2585] := 16#C3F5;
   // GB2[2586] := 16#C3F6;
   // GB2[2587] := 16#C3F7;
   // GB2[2588] := 16#C3F8;
   // GB2[2589] := 16#C3F9;
   // GB2[2590] := 16#C3FA;
   // GB2[2591] := 16#C3FB;
   // GB2[2592] := 16#C3FC;
   // GB2[2593] := 16#C3FD;
   // GB2[2594] := 16#C3FE;
   // GB2[2595] := 16#C4A1;
   // GB2[2596] := 16#C4A2;
   // GB2[2597] := 16#C4A3;
   // GB2[2598] := 16#C4A4;
   // GB2[2599] := 16#C4A5;
   // GB2[2600] := 16#C4A6;
   // GB2[2601] := 16#C4A7;
   // GB2[2602] := 16#C4A8;
   // GB2[2603] := 16#C4A9;
   // GB2[2604] := 16#C4AA;
   // GB2[2605] := 16#C4AB;
   // GB2[2606] := 16#C4AC;
   // GB2[2607] := 16#C4AD;
   // GB2[2608] := 16#C4AE;
   // GB2[2609] := 16#C4AF;
   // GB2[2610] := 16#C4B0;
   // GB2[2611] := 16#C4B1;
   // GB2[2612] := 16#C4B2;
   // GB2[2613] := 16#C4B3;
   // GB2[2614] := 16#C4B4;
   // GB2[2615] := 16#C4B5;
   // GB2[2616] := 16#C4B6;
   // GB2[2617] := 16#C4B7;
   // GB2[2618] := 16#C4B8;
   // GB2[2619] := 16#C4B9;
   // GB2[2620] := 16#C4BA;
   // GB2[2621] := 16#C4BB;
   // GB2[2622] := 16#C4BC;
   // GB2[2623] := 16#C4BD;
   // GB2[2624] := 16#C4BE;
   // GB2[2625] := 16#C4BF;
   // GB2[2626] := 16#C4C0;
   // GB2[2627] := 16#C4C1;
   // GB2[2628] := 16#C4C2;
   // GB2[2629] := 16#C4C3;
   // GB2[2630] := 16#C4C4;
   // GB2[2631] := 16#C4C5;
   // GB2[2632] := 16#C4C6;
   // GB2[2633] := 16#C4C7;
   // GB2[2634] := 16#C4C8;
   // GB2[2635] := 16#C4C9;
   // GB2[2636] := 16#C4CA;
   // GB2[2637] := 16#C4CB;
   // GB2[2638] := 16#C4CC;
   // GB2[2639] := 16#C4CD;
   // GB2[2640] := 16#C4CE;
   // GB2[2641] := 16#C4CF;
   // GB2[2642] := 16#C4D0;
   // GB2[2643] := 16#C4D1;
   // GB2[2644] := 16#C4D2;
   // GB2[2645] := 16#C4D3;
   // GB2[2646] := 16#C4D4;
   // GB2[2647] := 16#C4D5;
   // GB2[2648] := 16#C4D6;
   // GB2[2649] := 16#C4D7;
   // GB2[2650] := 16#C4D8;
   // GB2[2651] := 16#C4D9;
   // GB2[2652] := 16#C4DA;
   // GB2[2653] := 16#C4DB;
   // GB2[2654] := 16#C4DC;
   // GB2[2655] := 16#C4DD;
   // GB2[2656] := 16#C4DE;
   // GB2[2657] := 16#C4DF;
   // GB2[2658] := 16#C4E0;
   // GB2[2659] := 16#C4E1;
   // GB2[2660] := 16#C4E2;
   // GB2[2661] := 16#C4E3;
   // GB2[2662] := 16#C4E4;
   // GB2[2663] := 16#C4E5;
   // GB2[2664] := 16#C4E6;
   // GB2[2665] := 16#C4E7;
   // GB2[2666] := 16#C4E8;
   // GB2[2667] := 16#C4E9;
   // GB2[2668] := 16#C4EA;
   // GB2[2669] := 16#C4EB;
   // GB2[2670] := 16#C4EC;
   // GB2[2671] := 16#C4ED;
   // GB2[2672] := 16#C4EE;
   // GB2[2673] := 16#C4EF;
   // GB2[2674] := 16#C4F0;
   // GB2[2675] := 16#C4F1;
   // GB2[2676] := 16#C4F2;
   // GB2[2677] := 16#C4F3;
   // GB2[2678] := 16#C4F4;
   // GB2[2679] := 16#C4F5;
   // GB2[2680] := 16#C4F6;
   // GB2[2681] := 16#C4F7;
   // GB2[2682] := 16#C4F8;
   // GB2[2683] := 16#C4F9;
   // GB2[2684] := 16#C4FA;
   // GB2[2685] := 16#C4FB;
   // GB2[2686] := 16#C4FC;
   // GB2[2687] := 16#C4FD;
   // GB2[2688] := 16#C4FE;
   // GB2[2689] := 16#C5A1;
   // GB2[2690] := 16#C5A2;
   // GB2[2691] := 16#C5A3;
   // GB2[2692] := 16#C5A4;
   // GB2[2693] := 16#C5A5;
   // GB2[2694] := 16#C5A6;
   // GB2[2695] := 16#C5A7;
   // GB2[2696] := 16#C5A8;
   // GB2[2697] := 16#C5A9;
   // GB2[2698] := 16#C5AA;
   // GB2[2699] := 16#C5AB;
   // GB2[2700] := 16#C5AC;
   // GB2[2701] := 16#C5AD;
   // GB2[2702] := 16#C5AE;
   // GB2[2703] := 16#C5AF;
   // GB2[2704] := 16#C5B0;
   // GB2[2705] := 16#C5B1;
   // GB2[2706] := 16#C5B2;
   // GB2[2707] := 16#C5B3;
   // GB2[2708] := 16#C5B4;
   // GB2[2709] := 16#C5B5;
   // GB2[2710] := 16#C5B6;
   // GB2[2711] := 16#C5B7;
   // GB2[2712] := 16#C5B8;
   // GB2[2713] := 16#C5B9;
   // GB2[2714] := 16#C5BA;
   // GB2[2715] := 16#C5BB;
   // GB2[2716] := 16#C5BC;
   // GB2[2717] := 16#C5BD;
   // GB2[2718] := 16#C5BE;
   // GB2[2719] := 16#C5BF;
   // GB2[2720] := 16#C5C0;
   // GB2[2721] := 16#C5C1;
   // GB2[2722] := 16#C5C2;
   // GB2[2723] := 16#C5C3;
   // GB2[2724] := 16#C5C4;
   // GB2[2725] := 16#C5C5;
   // GB2[2726] := 16#C5C6;
   // GB2[2727] := 16#C5C7;
   // GB2[2728] := 16#C5C8;
   // GB2[2729] := 16#C5C9;
   // GB2[2730] := 16#C5CA;
   // GB2[2731] := 16#C5CB;
   // GB2[2732] := 16#C5CC;
   // GB2[2733] := 16#C5CD;
   // GB2[2734] := 16#C5CE;
   // GB2[2735] := 16#C5CF;
   // GB2[2736] := 16#C5D0;
   // GB2[2737] := 16#C5D1;
   // GB2[2738] := 16#C5D2;
   // GB2[2739] := 16#C5D3;
   // GB2[2740] := 16#C5D4;
   // GB2[2741] := 16#C5D5;
   // GB2[2742] := 16#C5D6;
   // GB2[2743] := 16#C5D7;
   // GB2[2744] := 16#C5D8;
   // GB2[2745] := 16#C5D9;
   // GB2[2746] := 16#C5DA;
   // GB2[2747] := 16#C5DB;
   // GB2[2748] := 16#C5DC;
   // GB2[2749] := 16#C5DD;
   // GB2[2750] := 16#C5DE;
   // GB2[2751] := 16#C5DF;
   // GB2[2752] := 16#C5E0;
   // GB2[2753] := 16#C5E1;
   // GB2[2754] := 16#C5E2;
   // GB2[2755] := 16#C5E3;
   // GB2[2756] := 16#C5E4;
   // GB2[2757] := 16#C5E5;
   // GB2[2758] := 16#C5E6;
   // GB2[2759] := 16#C5E7;
   // GB2[2760] := 16#C5E8;
   // GB2[2761] := 16#C5E9;
   // GB2[2762] := 16#C5EA;
   // GB2[2763] := 16#C5EB;
   // GB2[2764] := 16#C5EC;
   // GB2[2765] := 16#C5ED;
   // GB2[2766] := 16#C5EE;
   // GB2[2767] := 16#C5EF;
   // GB2[2768] := 16#C5F0;
   // GB2[2769] := 16#C5F1;
   // GB2[2770] := 16#C5F2;
   // GB2[2771] := 16#C5F3;
   // GB2[2772] := 16#C5F4;
   // GB2[2773] := 16#C5F5;
   // GB2[2774] := 16#C5F6;
   // GB2[2775] := 16#C5F7;
   // GB2[2776] := 16#C5F8;
   // GB2[2777] := 16#C5F9;
   // GB2[2778] := 16#C5FA;
   // GB2[2779] := 16#C5FB;
   // GB2[2780] := 16#C5FC;
   // GB2[2781] := 16#C5FD;
   // GB2[2782] := 16#C5FE;
   // GB2[2783] := 16#C6A1;
   // GB2[2784] := 16#C6A2;
   // GB2[2785] := 16#C6A3;
   // GB2[2786] := 16#C6A4;
   // GB2[2787] := 16#C6A5;
   // GB2[2788] := 16#C6A6;
   // GB2[2789] := 16#C6A7;
   // GB2[2790] := 16#C6A8;
   // GB2[2791] := 16#C6A9;
   // GB2[2792] := 16#C6AA;
   // GB2[2793] := 16#C6AB;
   // GB2[2794] := 16#C6AC;
   // GB2[2795] := 16#C6AD;
   // GB2[2796] := 16#C6AE;
   // GB2[2797] := 16#C6AF;
   // GB2[2798] := 16#C6B0;
   // GB2[2799] := 16#C6B1;
   // GB2[2800] := 16#C6B2;
   // GB2[2801] := 16#C6B3;
   // GB2[2802] := 16#C6B4;
   // GB2[2803] := 16#C6B5;
   // GB2[2804] := 16#C6B6;
   // GB2[2805] := 16#C6B7;
   // GB2[2806] := 16#C6B8;
   // GB2[2807] := 16#C6B9;
   // GB2[2808] := 16#C6BA;
   // GB2[2809] := 16#C6BB;
   // GB2[2810] := 16#C6BC;
   // GB2[2811] := 16#C6BD;
   // GB2[2812] := 16#C6BE;
   // GB2[2813] := 16#C6BF;
   // GB2[2814] := 16#C6C0;
   // GB2[2815] := 16#C6C1;
   // GB2[2816] := 16#C6C2;
   // GB2[2817] := 16#C6C3;
   // GB2[2818] := 16#C6C4;
   // GB2[2819] := 16#C6C5;
   // GB2[2820] := 16#C6C6;
   // GB2[2821] := 16#C6C7;
   // GB2[2822] := 16#C6C8;
   // GB2[2823] := 16#C6C9;
   // GB2[2824] := 16#C6CA;
   // GB2[2825] := 16#C6CB;
   // GB2[2826] := 16#C6CC;
   // GB2[2827] := 16#C6CD;
   // GB2[2828] := 16#C6CE;
   // GB2[2829] := 16#C6CF;
   // GB2[2830] := 16#C6D0;
   // GB2[2831] := 16#C6D1;
   // GB2[2832] := 16#C6D2;
   // GB2[2833] := 16#C6D3;
   // GB2[2834] := 16#C6D4;
   // GB2[2835] := 16#C6D5;
   // GB2[2836] := 16#C6D6;
   // GB2[2837] := 16#C6D7;
   // GB2[2838] := 16#C6D8;
   // GB2[2839] := 16#C6D9;
   // GB2[2840] := 16#C6DA;
   // GB2[2841] := 16#C6DB;
   // GB2[2842] := 16#C6DC;
   // GB2[2843] := 16#C6DD;
   // GB2[2844] := 16#C6DE;
   // GB2[2845] := 16#C6DF;
   // GB2[2846] := 16#C6E0;
   // GB2[2847] := 16#C6E1;
   // GB2[2848] := 16#C6E2;
   // GB2[2849] := 16#C6E3;
   // GB2[2850] := 16#C6E4;
   // GB2[2851] := 16#C6E5;
   // GB2[2852] := 16#C6E6;
   // GB2[2853] := 16#C6E7;
   // GB2[2854] := 16#C6E8;
   // GB2[2855] := 16#C6E9;
   // GB2[2856] := 16#C6EA;
   // GB2[2857] := 16#C6EB;
   // GB2[2858] := 16#C6EC;
   // GB2[2859] := 16#C6ED;
   // GB2[2860] := 16#C6EE;
   // GB2[2861] := 16#C6EF;
   // GB2[2862] := 16#C6F0;
   // GB2[2863] := 16#C6F1;
   // GB2[2864] := 16#C6F2;
   // GB2[2865] := 16#C6F3;
   // GB2[2866] := 16#C6F4;
   // GB2[2867] := 16#C6F5;
   // GB2[2868] := 16#C6F6;
   // GB2[2869] := 16#C6F7;
   // GB2[2870] := 16#C6F8;
   // GB2[2871] := 16#C6F9;
   // GB2[2872] := 16#C6FA;
   // GB2[2873] := 16#C6FB;
   // GB2[2874] := 16#C6FC;
   // GB2[2875] := 16#C6FD;
   // GB2[2876] := 16#C6FE;
   // GB2[2877] := 16#C7A1;
   // GB2[2878] := 16#C7A2;
   // GB2[2879] := 16#C7A3;
   // GB2[2880] := 16#C7A4;
   // GB2[2881] := 16#C7A5;
   // GB2[2882] := 16#C7A6;
   // GB2[2883] := 16#C7A7;
   // GB2[2884] := 16#C7A8;
   // GB2[2885] := 16#C7A9;
   // GB2[2886] := 16#C7AA;
   // GB2[2887] := 16#C7AB;
   // GB2[2888] := 16#C7AC;
   // GB2[2889] := 16#C7AD;
   // GB2[2890] := 16#C7AE;
   // GB2[2891] := 16#C7AF;
   // GB2[2892] := 16#C7B0;
   // GB2[2893] := 16#C7B1;
   // GB2[2894] := 16#C7B2;
   // GB2[2895] := 16#C7B3;
   // GB2[2896] := 16#C7B4;
   // GB2[2897] := 16#C7B5;
   // GB2[2898] := 16#C7B6;
   // GB2[2899] := 16#C7B7;
   // GB2[2900] := 16#C7B8;
   // GB2[2901] := 16#C7B9;
   // GB2[2902] := 16#C7BA;
   // GB2[2903] := 16#C7BB;
   // GB2[2904] := 16#C7BC;
   // GB2[2905] := 16#C7BD;
   // GB2[2906] := 16#C7BE;
   // GB2[2907] := 16#C7BF;
   // GB2[2908] := 16#C7C0;
   // GB2[2909] := 16#C7C1;
   // GB2[2910] := 16#C7C2;
   // GB2[2911] := 16#C7C3;
   // GB2[2912] := 16#C7C4;
   // GB2[2913] := 16#C7C5;
   // GB2[2914] := 16#C7C6;
   // GB2[2915] := 16#C7C7;
   // GB2[2916] := 16#C7C8;
   // GB2[2917] := 16#C7C9;
   // GB2[2918] := 16#C7CA;
   // GB2[2919] := 16#C7CB;
   // GB2[2920] := 16#C7CC;
   // GB2[2921] := 16#C7CD;
   // GB2[2922] := 16#C7CE;
   // GB2[2923] := 16#C7CF;
   // GB2[2924] := 16#C7D0;
   // GB2[2925] := 16#C7D1;
   // GB2[2926] := 16#C7D2;
   // GB2[2927] := 16#C7D3;
   // GB2[2928] := 16#C7D4;
   // GB2[2929] := 16#C7D5;
   // GB2[2930] := 16#C7D6;
   // GB2[2931] := 16#C7D7;
   // GB2[2932] := 16#C7D8;
   // GB2[2933] := 16#C7D9;
   // GB2[2934] := 16#C7DA;
   // GB2[2935] := 16#C7DB;
   // GB2[2936] := 16#C7DC;
   // GB2[2937] := 16#C7DD;
   // GB2[2938] := 16#C7DE;
   // GB2[2939] := 16#C7DF;
   // GB2[2940] := 16#C7E0;
   // GB2[2941] := 16#C7E1;
   // GB2[2942] := 16#C7E2;
   // GB2[2943] := 16#C7E3;
   // GB2[2944] := 16#C7E4;
   // GB2[2945] := 16#C7E5;
   // GB2[2946] := 16#C7E6;
   // GB2[2947] := 16#C7E7;
   // GB2[2948] := 16#C7E8;
   // GB2[2949] := 16#C7E9;
   // GB2[2950] := 16#C7EA;
   // GB2[2951] := 16#C7EB;
   // GB2[2952] := 16#C7EC;
   // GB2[2953] := 16#C7ED;
   // GB2[2954] := 16#C7EE;
   // GB2[2955] := 16#C7EF;
   // GB2[2956] := 16#C7F0;
   // GB2[2957] := 16#C7F1;
   // GB2[2958] := 16#C7F2;
   // GB2[2959] := 16#C7F3;
   // GB2[2960] := 16#C7F4;
   // GB2[2961] := 16#C7F5;
   // GB2[2962] := 16#C7F6;
   // GB2[2963] := 16#C7F7;
   // GB2[2964] := 16#C7F8;
   // GB2[2965] := 16#C7F9;
   // GB2[2966] := 16#C7FA;
   // GB2[2967] := 16#C7FB;
   // GB2[2968] := 16#C7FC;
   // GB2[2969] := 16#C7FD;
   // GB2[2970] := 16#C7FE;
   // GB2[2971] := 16#C8A1;
   // GB2[2972] := 16#C8A2;
   // GB2[2973] := 16#C8A3;
   // GB2[2974] := 16#C8A4;
   // GB2[2975] := 16#C8A5;
   // GB2[2976] := 16#C8A6;
   // GB2[2977] := 16#C8A7;
   // GB2[2978] := 16#C8A8;
   // GB2[2979] := 16#C8A9;
   // GB2[2980] := 16#C8AA;
   // GB2[2981] := 16#C8AB;
   // GB2[2982] := 16#C8AC;
   // GB2[2983] := 16#C8AD;
   // GB2[2984] := 16#C8AE;
   // GB2[2985] := 16#C8AF;
   // GB2[2986] := 16#C8B0;
   // GB2[2987] := 16#C8B1;
   // GB2[2988] := 16#C8B2;
   // GB2[2989] := 16#C8B3;
   // GB2[2990] := 16#C8B4;
   // GB2[2991] := 16#C8B5;
   // GB2[2992] := 16#C8B6;
   // GB2[2993] := 16#C8B7;
   // GB2[2994] := 16#C8B8;
   // GB2[2995] := 16#C8B9;
   // GB2[2996] := 16#C8BA;
   // GB2[2997] := 16#C8BB;
   // GB2[2998] := 16#C8BC;
   // GB2[2999] := 16#C8BD;
   // GB2[3000] := 16#C8BE;
   // GB2[3001] := 16#C8BF;
   // GB2[3002] := 16#C8C0;
   // GB2[3003] := 16#C8C1;
   // GB2[3004] := 16#C8C2;
   // GB2[3005] := 16#C8C3;
   // GB2[3006] := 16#C8C4;
   // GB2[3007] := 16#C8C5;
   // GB2[3008] := 16#C8C6;
   // GB2[3009] := 16#C8C7;
   // GB2[3010] := 16#C8C8;
   // GB2[3011] := 16#C8C9;
   // GB2[3012] := 16#C8CA;
   // GB2[3013] := 16#C8CB;
   // GB2[3014] := 16#C8CC;
   // GB2[3015] := 16#C8CD;
   // GB2[3016] := 16#C8CE;
   // GB2[3017] := 16#C8CF;
   // GB2[3018] := 16#C8D0;
   // GB2[3019] := 16#C8D1;
   // GB2[3020] := 16#C8D2;
   // GB2[3021] := 16#C8D3;
   // GB2[3022] := 16#C8D4;
   // GB2[3023] := 16#C8D5;
   // GB2[3024] := 16#C8D6;
   // GB2[3025] := 16#C8D7;
   // GB2[3026] := 16#C8D8;
   // GB2[3027] := 16#C8D9;
   // GB2[3028] := 16#C8DA;
   // GB2[3029] := 16#C8DB;
   // GB2[3030] := 16#C8DC;
   // GB2[3031] := 16#C8DD;
   // GB2[3032] := 16#C8DE;
   // GB2[3033] := 16#C8DF;
   // GB2[3034] := 16#C8E0;
   // GB2[3035] := 16#C8E1;
   // GB2[3036] := 16#C8E2;
   // GB2[3037] := 16#C8E3;
   // GB2[3038] := 16#C8E4;
   // GB2[3039] := 16#C8E5;
   // GB2[3040] := 16#C8E6;
   // GB2[3041] := 16#C8E7;
   // GB2[3042] := 16#C8E8;
   // GB2[3043] := 16#C8E9;
   // GB2[3044] := 16#C8EA;
   // GB2[3045] := 16#C8EB;
   // GB2[3046] := 16#C8EC;
   // GB2[3047] := 16#C8ED;
   // GB2[3048] := 16#C8EE;
   // GB2[3049] := 16#C8EF;
   // GB2[3050] := 16#C8F0;
   // GB2[3051] := 16#C8F1;
   // GB2[3052] := 16#C8F2;
   // GB2[3053] := 16#C8F3;
   // GB2[3054] := 16#C8F4;
   // GB2[3055] := 16#C8F5;
   // GB2[3056] := 16#C8F6;
   // GB2[3057] := 16#C8F7;
   // GB2[3058] := 16#C8F8;
   // GB2[3059] := 16#C8F9;
   // GB2[3060] := 16#C8FA;
   // GB2[3061] := 16#C8FB;
   // GB2[3062] := 16#C8FC;
   // GB2[3063] := 16#C8FD;
   // GB2[3064] := 16#C8FE;
   // GB2[3065] := 16#C9A1;
   // GB2[3066] := 16#C9A2;
   // GB2[3067] := 16#C9A3;
   // GB2[3068] := 16#C9A4;
   // GB2[3069] := 16#C9A5;
   // GB2[3070] := 16#C9A6;
   // GB2[3071] := 16#C9A7;
   // GB2[3072] := 16#C9A8;
   // GB2[3073] := 16#C9A9;
   // GB2[3074] := 16#C9AA;
   // GB2[3075] := 16#C9AB;
   // GB2[3076] := 16#C9AC;
   // GB2[3077] := 16#C9AD;
   // GB2[3078] := 16#C9AE;
   // GB2[3079] := 16#C9AF;
   // GB2[3080] := 16#C9B0;
   // GB2[3081] := 16#C9B1;
   // GB2[3082] := 16#C9B2;
   // GB2[3083] := 16#C9B3;
   // GB2[3084] := 16#C9B4;
   // GB2[3085] := 16#C9B5;
   // GB2[3086] := 16#C9B6;
   // GB2[3087] := 16#C9B7;
   // GB2[3088] := 16#C9B8;
   // GB2[3089] := 16#C9B9;
   // GB2[3090] := 16#C9BA;
   // GB2[3091] := 16#C9BB;
   // GB2[3092] := 16#C9BC;
   // GB2[3093] := 16#C9BD;
   // GB2[3094] := 16#C9BE;
   // GB2[3095] := 16#C9BF;
   // GB2[3096] := 16#C9C0;
   // GB2[3097] := 16#C9C1;
   // GB2[3098] := 16#C9C2;
   // GB2[3099] := 16#C9C3;
   // GB2[3100] := 16#C9C4;
   // GB2[3101] := 16#C9C5;
   // GB2[3102] := 16#C9C6;
   // GB2[3103] := 16#C9C7;
   // GB2[3104] := 16#C9C8;
   // GB2[3105] := 16#C9C9;
   // GB2[3106] := 16#C9CA;
   // GB2[3107] := 16#C9CB;
   // GB2[3108] := 16#C9CC;
   // GB2[3109] := 16#C9CD;
   // GB2[3110] := 16#C9CE;
   // GB2[3111] := 16#C9CF;
   // GB2[3112] := 16#C9D0;
   // GB2[3113] := 16#C9D1;
   // GB2[3114] := 16#C9D2;
   // GB2[3115] := 16#C9D3;
   // GB2[3116] := 16#C9D4;
   // GB2[3117] := 16#C9D5;
   // GB2[3118] := 16#C9D6;
   // GB2[3119] := 16#C9D7;
   // GB2[3120] := 16#C9D8;
   // GB2[3121] := 16#C9D9;
   // GB2[3122] := 16#C9DA;
   // GB2[3123] := 16#C9DB;
   // GB2[3124] := 16#C9DC;
   // GB2[3125] := 16#C9DD;
   // GB2[3126] := 16#C9DE;
   // GB2[3127] := 16#C9DF;
   // GB2[3128] := 16#C9E0;
   // GB2[3129] := 16#C9E1;
   // GB2[3130] := 16#C9E2;
   // GB2[3131] := 16#C9E3;
   // GB2[3132] := 16#C9E4;
   // GB2[3133] := 16#C9E5;
   // GB2[3134] := 16#C9E6;
   // GB2[3135] := 16#C9E7;
   // GB2[3136] := 16#C9E8;
   // GB2[3137] := 16#C9E9;
   // GB2[3138] := 16#C9EA;
   // GB2[3139] := 16#C9EB;
   // GB2[3140] := 16#C9EC;
   // GB2[3141] := 16#C9ED;
   // GB2[3142] := 16#C9EE;
   // GB2[3143] := 16#C9EF;
   // GB2[3144] := 16#C9F0;
   // GB2[3145] := 16#C9F1;
   // GB2[3146] := 16#C9F2;
   // GB2[3147] := 16#C9F3;
   // GB2[3148] := 16#C9F4;
   // GB2[3149] := 16#C9F5;
   // GB2[3150] := 16#C9F6;
   // GB2[3151] := 16#C9F7;
   // GB2[3152] := 16#C9F8;
   // GB2[3153] := 16#C9F9;
   // GB2[3154] := 16#C9FA;
   // GB2[3155] := 16#C9FB;
   // GB2[3156] := 16#C9FC;
   // GB2[3157] := 16#C9FD;
   // GB2[3158] := 16#C9FE;
   // GB2[3159] := 16#CAA1;
   // GB2[3160] := 16#CAA2;
   // GB2[3161] := 16#CAA3;
   // GB2[3162] := 16#CAA4;
   // GB2[3163] := 16#CAA5;
   // GB2[3164] := 16#CAA6;
   // GB2[3165] := 16#CAA7;
   // GB2[3166] := 16#CAA8;
   // GB2[3167] := 16#CAA9;
   // GB2[3168] := 16#CAAA;
   // GB2[3169] := 16#CAAB;
   // GB2[3170] := 16#CAAC;
   // GB2[3171] := 16#CAAD;
   // GB2[3172] := 16#CAAE;
   // GB2[3173] := 16#CAAF;
   // GB2[3174] := 16#CAB0;
   // GB2[3175] := 16#CAB1;
   // GB2[3176] := 16#CAB2;
   // GB2[3177] := 16#CAB3;
   // GB2[3178] := 16#CAB4;
   // GB2[3179] := 16#CAB5;
   // GB2[3180] := 16#CAB6;
   // GB2[3181] := 16#CAB7;
   // GB2[3182] := 16#CAB8;
   // GB2[3183] := 16#CAB9;
   // GB2[3184] := 16#CABA;
   // GB2[3185] := 16#CABB;
   // GB2[3186] := 16#CABC;
   // GB2[3187] := 16#CABD;
   // GB2[3188] := 16#CABE;
   // GB2[3189] := 16#CABF;
   // GB2[3190] := 16#CAC0;
   // GB2[3191] := 16#CAC1;
   // GB2[3192] := 16#CAC2;
   // GB2[3193] := 16#CAC3;
   // GB2[3194] := 16#CAC4;
   // GB2[3195] := 16#CAC5;
   // GB2[3196] := 16#CAC6;
   // GB2[3197] := 16#CAC7;
   // GB2[3198] := 16#CAC8;
   // GB2[3199] := 16#CAC9;
   // GB2[3200] := 16#CACA;
   // GB2[3201] := 16#CACB;
   // GB2[3202] := 16#CACC;
   // GB2[3203] := 16#CACD;
   // GB2[3204] := 16#CACE;
   // GB2[3205] := 16#CACF;
   // GB2[3206] := 16#CAD0;
   // GB2[3207] := 16#CAD1;
   // GB2[3208] := 16#CAD2;
   // GB2[3209] := 16#CAD3;
   // GB2[3210] := 16#CAD4;
   // GB2[3211] := 16#CAD5;
   // GB2[3212] := 16#CAD6;
   // GB2[3213] := 16#CAD7;
   // GB2[3214] := 16#CAD8;
   // GB2[3215] := 16#CAD9;
   // GB2[3216] := 16#CADA;
   // GB2[3217] := 16#CADB;
   // GB2[3218] := 16#CADC;
   // GB2[3219] := 16#CADD;
   // GB2[3220] := 16#CADE;
   // GB2[3221] := 16#CADF;
   // GB2[3222] := 16#CAE0;
   // GB2[3223] := 16#CAE1;
   // GB2[3224] := 16#CAE2;
   // GB2[3225] := 16#CAE3;
   // GB2[3226] := 16#CAE4;
